// mobject-converters/Converters/REAL_TO_/TryConvert_REAL_TO_UINT
FUNCTION TryConvert_REAL_TO_UINT : BOOL
VAR_INPUT
	in : REAL;
	out : REFERENCE TO UINT;
END_VAR

IF in > DatatypeLimits.MAX_VALUE_OF_REAL_WHICH_CAN_BE_HELD_IN_A_UINT THEN
	RETURN;
END_IF

IF in < DatatypeLimits.MIN_VALUE_OF_REAL_WHICH_CAN_BE_HELD_IN_A_UINT THEN
	RETURN;
END_IF

out := REAL_TO_UINT(in);
TryConvert_REAL_TO_UINT := TRUE;

END_FUNCTION

// mobject-converters/Converters/REAL_TO_/TryConvert_REAL_TO_UDINT
FUNCTION TryConvert_REAL_TO_UDINT : BOOL
VAR_INPUT
	in : REAL;
	out : REFERENCE TO UDINT;
END_VAR

IF in > DatatypeLimits.MAX_VALUE_OF_REAL_WHICH_CAN_BE_HELD_IN_A_UDINT THEN
	RETURN;
END_IF

IF in < DatatypeLimits.MIN_VALUE_OF_REAL_WHICH_CAN_BE_HELD_IN_A_UDINT THEN
	RETURN;
END_IF

out := REAL_TO_UDINT(in);
TryConvert_REAL_TO_UDINT := TRUE;

END_FUNCTION

// mobject-converters/Converters/REAL_TO_/TryConvert_REAL_TO_ULINT
FUNCTION TryConvert_REAL_TO_ULINT : BOOL
VAR_INPUT
	in : REAL;
	out : REFERENCE TO ULINT;
END_VAR

IF in > DatatypeLimits.MAX_VALUE_OF_REAL_WHICH_CAN_BE_HELD_IN_A_ULINT THEN
	RETURN;
END_IF

IF in < DatatypeLimits.MIN_VALUE_OF_REAL_WHICH_CAN_BE_HELD_IN_A_ULINT THEN
	RETURN;
END_IF

out := REAL_TO_ULINT(in);
TryConvert_REAL_TO_ULINT := TRUE;

END_FUNCTION

// mobject-converters/Converters/REAL_TO_/TryConvert_REAL_TO_REAL
FUNCTION TryConvert_REAL_TO_REAL : BOOL
VAR_INPUT
	in : REAL;
	out : REFERENCE TO REAL;
END_VAR

out := in;
TryConvert_REAL_TO_REAL := TRUE;

END_FUNCTION

// mobject-converters/Converters/REAL_TO_/TryConvert_REAL_TO_LREAL
FUNCTION TryConvert_REAL_TO_LREAL : BOOL
VAR_INPUT
	in : REAL;
	out : REFERENCE TO LREAL;
END_VAR

out := REAL_TO_LREAL(in);
TryConvert_REAL_TO_LREAL := TRUE;

END_FUNCTION

// mobject-datatypes/Primitive/_LREAL
{attribute 'linkalways'} 
{attribute 'no_explicit_call' := 'This FB is a CLASS and must be accessed using methods or properties'}
{attribute 'enable_dynamic_creation'}
FUNCTION_BLOCK _LREAL EXTENDS NumericDatatypeBase IMPLEMENTS I_LREAL
VAR
	localData : LREAL;
	activeData : REFERENCE TO LREAL REF= localData;
END_VAR

METHOD FB_init : BOOL
VAR_INPUT
	bInitRetains : BOOL; // if TRUE, the retain variables are initialized (warm start / cold start)
	bInCopyCode : BOOL;  // if TRUE, the instance afterwards gets moved into the copy code (online change)
	InitialValue : LREAL;
END_VAR
localData := InitialValue;
END_METHOD

METHOD PROTECTED SerializeMaxValue
VAR_INPUT
	Serializer : I_Serializer;
END_VAR
Serializer.AddLreal(MaxValue);
END_METHOD

METHOD PROTECTED SerializeMinValue
VAR_INPUT
	Serializer : I_Serializer;
END_VAR
Serializer.AddLreal(MinValue);
END_METHOD

PROPERTY PUBLIC Address : PVOID
GET
Address := ADR(activeData);
END_GET
END_PROPERTY

METHOD PUBLIC ClearReference
VAR_INPUT
END_VAR
activeData REF= localData;
END_METHOD

METHOD PUBLIC Clone : I_Datatype
VAR
    pClone : POINTER TO _LREAL;
END_VAR
pClone := __NEW(_LREAL(InitialValue := Value));
Clone := pClone^;
END_METHOD

PROPERTY PUBLIC IsEven : BOOL
GET
IsEven := FALSE;
END_GET
END_PROPERTY

PROPERTY PUBLIC IsFloat : BOOL
GET
IsFloat := TRUE;
END_GET
END_PROPERTY

PROPERTY PUBLIC IsOdd : BOOL
GET
IsOdd := FALSE;
END_GET
END_PROPERTY

PROPERTY PUBLIC IsSigned : BOOL
GET
IsSigned := TRUE;
END_GET
END_PROPERTY

METHOD PUBLIC MakeReferenceTo
VAR_INPUT
	ReferenceTarget : REFERENCE TO LREAL;
END_VAR
activeData REF= ReferenceTarget;
END_METHOD

PROPERTY PUBLIC MaxValue : LREAL
GET
MaxValue :=  DatatypeLimits.LREAL_MAX_VALUE;
END_GET
END_PROPERTY

PROPERTY PUBLIC MinValue : LREAL
GET
MinValue := DatatypeLimits.LREAL_MIN_VALUE;
END_GET
END_PROPERTY

METHOD PUBLIC SerializeWith
VAR_INPUT
	Serializer : I_Serializer;
END_VAR
Serializer.AddLreal(activeData);
END_METHOD

PROPERTY PUBLIC Size : UDINT
GET
Size := SIZEOF(activeData);
END_GET
END_PROPERTY

METHOD PUBLIC TryConvertTo : BOOL
VAR_INPUT
	Destination : ANY;
END_VAR
TryConvertTo := TryConvert_LREAL_To_Destination(activeData, Destination);
END_METHOD

METHOD PUBLIC TryConvertTo_ : BOOL
VAR_INPUT
	Destination : I_Datatype;
END_VAR
VAR
	resultofBitConversion : BOOL;
	destinationAs_BIT : I_BIT;
	destinationAs_BOOL : I_BOOL;
	destinationAs_BYTE : I_BYTE;
	destinationAs_DINT : I_DINT;
	destinationAs_DT : I_DT;
	destinationAs_DWORD : I_DWORD;
	destinationAs_INT : I_INT;
	destinationAs_LINT : I_LINT;
	destinationAs_LREAL : I_LREAL;
	destinationAs_LWORD : I_LWORD;
	destinationAs_REAL : I_REAL;
	destinationAs_SINT : I_SINT;
	destinationAs_STRING : I_STRING;
	destinationAs_TOD : I_TOD;
	destinationAs_UDINT : I_UDINT;
	destinationAs_UINT : I_UINT;
	destinationAs_ULINT : I_ULINT;
	destinationAs_USINT : I_USINT;
	destinationAs_WORD : I_WORD;
END_VAR
IF destination.TryResolveAs_BIT(destinationAs_BIT) AND_THEN TryConvert_LREAL_TO_BOOL(activeData, resultofBitConversion) THEN
	destinationAs_BIT.Value := resultOfBitConversion;
	TryConvertTo_ := TRUE;
	RETURN;
END_IF

IF destination.TryResolveAs_BOOL(destinationAs_BOOL) THEN
	TryConvertTo_ := TryConvert_LREAL_TO_BOOL(activeData, destinationAs_BOOL.Value);
	RETURN;
END_IF
		
IF destination.TryResolveAs_BYTE(destinationAs_BYTE) THEN
	TryConvertTo_ := TryConvert_LREAL_TO_BYTE(activeData, destinationAs_BYTE.Value);
	RETURN;
END_IF

IF destination.TryResolveAs_DINT(destinationAs_DINT) THEN
	TryConvertTo_ := TryConvert_LREAL_TO_DINT(activeData, destinationAs_DINT.Value);
	RETURN;
END_IF

IF destination.TryResolveAs_DT(destinationAs_DT) THEN
	TryConvertTo_ := TryConvert_LREAL_TO_DT(activeData, destinationAs_DT.Value);
	RETURN;
END_IF

IF destination.TryResolveAs_DWORD(destinationAs_DWORD) THEN
	TryConvertTo_ := TryConvert_LREAL_TO_DWORD(activeData, destinationAs_DWORD.Value);
	RETURN;
END_IF

IF destination.TryResolveAs_INT(destinationAs_INT) THEN
	TryConvertTo_ := TryConvert_LREAL_TO_INT(activeData, destinationAs_INT.Value);
	RETURN;
END_IF

IF destination.TryResolveAs_LINT(destinationAs_LINT) THEN
	TryConvertTo_ := TryConvert_LREAL_TO_LINT(activeData, destinationAs_LINT.Value);
	RETURN;
END_IF

IF destination.TryResolveAs_LREAL(destinationAs_LREAL) THEN
	TryConvertTo_ := TryConvert_LREAL_TO_LREAL(activeData, destinationAs_LREAL.Value);
	RETURN;
END_IF

IF destination.TryResolveAs_LWORD(destinationAs_LWORD) THEN
	TryConvertTo_ := TryConvert_LREAL_TO_LWORD(activeData, destinationAs_LWORD.Value);
	RETURN;
END_IF

IF destination.TryResolveAs_REAL(destinationAs_REAL) THEN
	TryConvertTo_ := TryConvert_LREAL_TO_REAL(activeData, destinationAs_REAL.Value);
	RETURN;
END_IF

IF destination.TryResolveAs_SINT(destinationAs_SINT) THEN
	TryConvertTo_ := TryConvert_LREAL_TO_SINT(activeData, destinationAs_SINT.Value);
	RETURN;
END_IF

IF destination.TryResolveAs_STRING(destinationAs_STRING) THEN
	TryConvertTo_ := TryConvert_LREAL_TO_STRING(activeData, destinationAs_STRING.Value);
	RETURN;
END_IF

IF destination.TryResolveAs_TOD(destinationAs_TOD) THEN
	TryConvertTo_ := TryConvert_LREAL_TO_TOD(activeData, destinationAs_TOD.Value);
	RETURN;
END_IF

IF destination.TryResolveAs_UDINT(destinationAs_UDINT) THEN
	TryConvertTo_ := TryConvert_LREAL_TO_UDINT(activeData, destinationAs_UDINT.Value);
	RETURN;
END_IF

IF destination.TryResolveAs_UINT(destinationAs_UINT) THEN
	TryConvertTo_ := TryConvert_LREAL_TO_UINT(activeData, destinationAs_UINT.Value);
	RETURN;
END_IF

IF destination.TryResolveAs_ULINT(destinationAs_ULINT) THEN
	TryConvertTo_ := TryConvert_LREAL_TO_ULINT(activeData, destinationAs_ULINT.Value);
	RETURN;
END_IF

IF destination.TryResolveAs_USINT(destinationAs_USINT) THEN
	TryConvertTo_ := TryConvert_LREAL_TO_USINT(activeData, destinationAs_USINT.Value);
	RETURN;
END_IF

IF destination.TryResolveAs_WORD(destinationAs_WORD) THEN
	TryConvertTo_ := TryConvert_LREAL_TO_WORD(activeData, destinationAs_WORD.Value);
	RETURN;
END_IF
END_METHOD

METHOD TryDeserializeFrom : BOOL
VAR_INPUT
	Deserializer : I_Deserializer;
	Feedback : I_DeserializerFeedback;
END_VAR
TryDeserializeFrom := Deserializer.TryGetLreal(activeData, Feedback);
END_METHOD

METHOD TryMakeReferenceTo : BOOL
VAR_INPUT
	Target : I_Datatype;
END_VAR
VAR
	pTargetData : POINTER TO LREAL;
END_VAR
IF NOT IsEquivalentTo(Target) THEN
	RETURN;
END_IF

pTargetData := Target.Address;
activeData REF= pTargetData^;
TryMakeReferenceTo := TRUE;
END_METHOD

METHOD PUBLIC TryResolveAs_LREAL : BOOL
VAR_INPUT
	Destination : REFERENCE TO I_LREAL;
END_VAR
Destination := THIS^;
TryResolveAs_LREAL := TRUE;
END_METHOD

PROPERTY PUBLIC TypeName : T_MAXSTRING
GET
TypeName := 'LREAL';
END_GET
END_PROPERTY

{warning disable C5410}
PROPERTY PUBLIC Value : REFERENCE TO LREAL
{warning restore C5410}
GET
Value REF= activeData;
END_GET
END_PROPERTY

END_FUNCTION_BLOCK

// mobject-converters/Converters/LREAL_TO_/TryConvert_LREAL_TO_Destination
FUNCTION TryConvert_LREAL_TO_Destination : BOOL
VAR_INPUT
	in : LREAL;
	out : ANY;
END_VAR
VAR
	convertResult : BOOL := FALSE;
	convertAddress : PVOID;
	_BOOL : BOOL;
	_BYTE : BYTE;
	_WORD : WORD;
	_DWORD : DWORD;
	_LWORD : LWORD;
	_SINT : SINT;
	_INT : INT;
	_DINT : DINT;
	_LINT : LINT;
	_USINT : USINT;
	_UINT : UINT;
	_UDINT : UDINT;
	_ULINT : ULINT;
	_REAL : REAL;
	_LREAL : LREAL;
	_TIME : TIME;
	_TOD : TOD;
	_DATE : DATE;
	_DT : DT;
	_STRING : STRING;
END_VAR

CASE out.TypeClass OF
	__SYSTEM.TYPE_CLASS.TYPE_BOOL:
	
	convertResult := TryConvert_LREAL_TO_BOOL(in, _BOOL);
	IF convertResult THEN
		convertAddress := ADR(_BOOL);
	END_IF
	
	__SYSTEM.TYPE_CLASS.TYPE_BYTE:
	
	convertResult := TryConvert_LREAL_TO_BYTE(in, _BYTE);
	IF convertResult THEN
		convertAddress := ADR(_BYTE);
	END_IF
	
	__SYSTEM.TYPE_CLASS.TYPE_WORD:
	
	convertResult := TryConvert_LREAL_TO_WORD(in, _WORD);
	IF convertResult THEN
		convertAddress := ADR(_WORD);
	END_IF
	
	__SYSTEM.TYPE_CLASS.TYPE_DWORD:
	
	convertResult := TryConvert_LREAL_TO_DWORD(in, _DWORD);
	IF convertResult THEN
		convertAddress := ADR(_DWORD);
	END_IF
	
	__SYSTEM.TYPE_CLASS.TYPE_LWORD:
	
	convertResult := TryConvert_LREAL_TO_LWORD(in, _LWORD);
	IF convertResult THEN
		convertAddress := ADR(_LWORD);
	END_IF
	
	__SYSTEM.TYPE_CLASS.TYPE_SINT:
	
	convertResult := TryConvert_LREAL_TO_SINT(in, _SINT);
	IF convertResult THEN
		convertAddress := ADR(_SINT);
	END_IF
	
	__SYSTEM.TYPE_CLASS.TYPE_INT:
	
	convertResult := TryConvert_LREAL_TO_INT(in, _INT);
	IF convertResult THEN
		convertAddress := ADR(_INT);
	END_IF
	
	__SYSTEM.TYPE_CLASS.TYPE_DINT:
	
	convertResult := TryConvert_LREAL_TO_DINT(in, _DINT);
	IF convertResult THEN
		convertAddress := ADR(_DINT);
	END_IF
	
	__SYSTEM.TYPE_CLASS.TYPE_LINT:
	
	convertResult := TryConvert_LREAL_TO_LINT(in, _LINT);
	IF convertResult THEN
		convertAddress := ADR(_LINT);
	END_IF
	
	__SYSTEM.TYPE_CLASS.TYPE_USINT:
	
	convertResult := TryConvert_LREAL_TO_USINT(in, _USINT);
	IF convertResult THEN
		convertAddress := ADR(_USINT);
	END_IF
	
	__SYSTEM.TYPE_CLASS.TYPE_UINT:
	
	convertResult := TryConvert_LREAL_TO_UINT(in, _UINT);
	IF convertResult THEN
		convertAddress := ADR(_UINT);
	END_IF
	
	__SYSTEM.TYPE_CLASS.TYPE_UDINT:
	
	convertResult := TryConvert_LREAL_TO_UDINT(in, _UDINT);
	IF convertResult THEN
		convertAddress := ADR(_UDINT);
	END_IF
	
	__SYSTEM.TYPE_CLASS.TYPE_ULINT:
	
	convertResult := TryConvert_LREAL_TO_ULINT(in, _ULINT);
	IF convertResult THEN
		convertAddress := ADR(_ULINT);
	END_IF
	
	__SYSTEM.TYPE_CLASS.TYPE_REAL:
	
	convertResult := TryConvert_LREAL_TO_REAL(in, _REAL);
	IF convertResult THEN
		convertAddress := ADR(_REAL);
	END_IF
	
	__SYSTEM.TYPE_CLASS.TYPE_LREAL:
	
	convertResult := TryConvert_LREAL_TO_LREAL(in, _LREAL);
	IF convertResult THEN
		convertAddress := ADR(_LREAL);
	END_IF
	
	__SYSTEM.TYPE_CLASS.TYPE_TIME:
	
	convertResult := TryConvert_LREAL_TO_TIME(in, _TIME);
	IF convertResult THEN
		convertAddress := ADR(_TIME);
	END_IF
	
	__SYSTEM.TYPE_CLASS.TYPE_TIMEOFDAY:
	
	convertResult := TryConvert_LREAL_TO_TOD(in, _TOD);
	IF convertResult THEN
		convertAddress := ADR(_TOD);
	END_IF
	
	__SYSTEM.TYPE_CLASS.TYPE_DATE:
	
	convertResult := TryConvert_LREAL_TO_DATE(in, _DATE);
	IF convertResult THEN
		convertAddress := ADR(_DATE);
	END_IF
	
	__SYSTEM.TYPE_CLASS.TYPE_DATEANDTIME:
	
	convertResult := TryConvert_LREAL_TO_DT(in, _DT);
	IF convertResult THEN
		convertAddress := ADR(_DT);
	END_IF
	
	__SYSTEM.TYPE_CLASS.TYPE_STRING:
	
	convertResult := TryConvert_LREAL_TO_STRING(in, _STRING);
	IF convertResult THEN
		convertAddress := ADR(_STRING);
	END_IF
	
END_CASE

IF convertResult THEN
	memcpy(out.pValue,convertAddress,DINT_TO_UDINT(out.diSize));
END_IF

TryConvert_LREAL_TO_Destination := convertResult;

END_FUNCTION

// mobject-converters/Converters/LREAL_TO_/TryConvert_LREAL_TO_BOOL
FUNCTION TryConvert_LREAL_TO_BOOL : BOOL
VAR_INPUT
	in : LREAL;
	out : REFERENCE TO BOOL;
END_VAR

out := LREAL_TO_BOOL(in);
TryConvert_LREAL_TO_BOOL := TRUE;

END_FUNCTION

// mobject-converters/Converters/LREAL_TO_/TryConvert_LREAL_TO_BYTE
FUNCTION TryConvert_LREAL_TO_BYTE : BOOL
VAR_INPUT
	in : LREAL;
	out : REFERENCE TO BYTE;
END_VAR

IF in > DatatypeLimits.MAX_VALUE_OF_LREAL_WHICH_CAN_BE_HELD_IN_A_BYTE THEN
	RETURN;
END_IF

IF in < DatatypeLimits.MIN_VALUE_OF_LREAL_WHICH_CAN_BE_HELD_IN_A_BYTE THEN
	RETURN;
END_IF

out := LREAL_TO_BYTE(in);
TryConvert_LREAL_TO_BYTE := TRUE;

END_FUNCTION

// mobject-converters/Converters/LREAL_TO_/TryConvert_LREAL_TO_WORD
FUNCTION TryConvert_LREAL_TO_WORD : BOOL
VAR_INPUT
	in : LREAL;
	out : REFERENCE TO WORD;
END_VAR

IF in > DatatypeLimits.MAX_VALUE_OF_LREAL_WHICH_CAN_BE_HELD_IN_A_WORD THEN
	RETURN;
END_IF

IF in < DatatypeLimits.MIN_VALUE_OF_LREAL_WHICH_CAN_BE_HELD_IN_A_WORD THEN
	RETURN;
END_IF

out := LREAL_TO_WORD(in);
TryConvert_LREAL_TO_WORD := TRUE;

END_FUNCTION

// mobject-converters/Converters/LREAL_TO_/TryConvert_LREAL_TO_DWORD
FUNCTION TryConvert_LREAL_TO_DWORD : BOOL
VAR_INPUT
	in : LREAL;
	out : REFERENCE TO DWORD;
END_VAR

IF in > DatatypeLimits.MAX_VALUE_OF_LREAL_WHICH_CAN_BE_HELD_IN_A_DWORD THEN
	RETURN;
END_IF

IF in < DatatypeLimits.MIN_VALUE_OF_LREAL_WHICH_CAN_BE_HELD_IN_A_DWORD THEN
	RETURN;
END_IF

out := LREAL_TO_DWORD(in);
TryConvert_LREAL_TO_DWORD := TRUE;

END_FUNCTION

// mobject-converters/Converters/LREAL_TO_/TryConvert_LREAL_TO_LWORD
FUNCTION TryConvert_LREAL_TO_LWORD : BOOL
VAR_INPUT
	in : LREAL;
	out : REFERENCE TO LWORD;
END_VAR

IF in > DatatypeLimits.MAX_VALUE_OF_LREAL_WHICH_CAN_BE_HELD_IN_A_LWORD THEN
	RETURN;
END_IF

IF in < DatatypeLimits.MIN_VALUE_OF_LREAL_WHICH_CAN_BE_HELD_IN_A_LWORD THEN
	RETURN;
END_IF

out := LREAL_TO_LWORD(in);
TryConvert_LREAL_TO_LWORD := TRUE;

END_FUNCTION

// mobject-converters/Converters/LREAL_TO_/TryConvert_LREAL_TO_SINT
FUNCTION TryConvert_LREAL_TO_SINT : BOOL
VAR_INPUT
	in : LREAL;
	out : REFERENCE TO SINT;
END_VAR

IF in > DatatypeLimits.MAX_VALUE_OF_LREAL_WHICH_CAN_BE_HELD_IN_A_SINT THEN
	RETURN;
END_IF

IF in < DatatypeLimits.MIN_VALUE_OF_LREAL_WHICH_CAN_BE_HELD_IN_A_SINT THEN
	RETURN;
END_IF

out := LREAL_TO_SINT(in);
TryConvert_LREAL_TO_SINT := TRUE;

END_FUNCTION

// mobject-converters/Converters/LREAL_TO_/TryConvert_LREAL_TO_INT
FUNCTION TryConvert_LREAL_TO_INT : BOOL
VAR_INPUT
	in : LREAL;
	out : REFERENCE TO INT;
END_VAR

IF in > DatatypeLimits.MAX_VALUE_OF_LREAL_WHICH_CAN_BE_HELD_IN_A_INT THEN
	RETURN;
END_IF

IF in < DatatypeLimits.MIN_VALUE_OF_LREAL_WHICH_CAN_BE_HELD_IN_A_INT THEN
	RETURN;
END_IF

out := LREAL_TO_INT(in);
TryConvert_LREAL_TO_INT := TRUE;

END_FUNCTION

// mobject-converters/Converters/LREAL_TO_/TryConvert_LREAL_TO_DINT
FUNCTION TryConvert_LREAL_TO_DINT : BOOL
VAR_INPUT
	in : LREAL;
	out : REFERENCE TO DINT;
END_VAR

IF in > DatatypeLimits.MAX_VALUE_OF_LREAL_WHICH_CAN_BE_HELD_IN_A_DINT THEN
	RETURN;
END_IF

IF in < DatatypeLimits.MIN_VALUE_OF_LREAL_WHICH_CAN_BE_HELD_IN_A_DINT THEN
	RETURN;
END_IF

out := LREAL_TO_DINT(in);
TryConvert_LREAL_TO_DINT := TRUE;

END_FUNCTION

// mobject-converters/Converters/LREAL_TO_/TryConvert_LREAL_TO_LINT
FUNCTION TryConvert_LREAL_TO_LINT : BOOL
VAR_INPUT
	in : LREAL;
	out : REFERENCE TO LINT;
END_VAR

IF in > DatatypeLimits.MAX_VALUE_OF_LREAL_WHICH_CAN_BE_HELD_IN_A_LINT THEN
	RETURN;
END_IF

IF in < DatatypeLimits.MIN_VALUE_OF_LREAL_WHICH_CAN_BE_HELD_IN_A_LINT THEN
	RETURN;
END_IF

out := LREAL_TO_LINT(in);
TryConvert_LREAL_TO_LINT := TRUE;

END_FUNCTION

// mobject-converters/Converters/LREAL_TO_/TryConvert_LREAL_TO_USINT
FUNCTION TryConvert_LREAL_TO_USINT : BOOL
VAR_INPUT
	in : LREAL;
	out : REFERENCE TO USINT;
END_VAR

IF in > DatatypeLimits.MAX_VALUE_OF_LREAL_WHICH_CAN_BE_HELD_IN_A_USINT THEN
	RETURN;
END_IF

IF in < DatatypeLimits.MIN_VALUE_OF_LREAL_WHICH_CAN_BE_HELD_IN_A_USINT THEN
	RETURN;
END_IF

out := LREAL_TO_USINT(in);
TryConvert_LREAL_TO_USINT := TRUE;

END_FUNCTION

// mobject-converters/Converters/LREAL_TO_/TryConvert_LREAL_TO_UINT
FUNCTION TryConvert_LREAL_TO_UINT : BOOL
VAR_INPUT
	in : LREAL;
	out : REFERENCE TO UINT;
END_VAR

IF in > DatatypeLimits.MAX_VALUE_OF_LREAL_WHICH_CAN_BE_HELD_IN_A_UINT THEN
	RETURN;
END_IF

IF in < DatatypeLimits.MIN_VALUE_OF_LREAL_WHICH_CAN_BE_HELD_IN_A_UINT THEN
	RETURN;
END_IF

out := LREAL_TO_UINT(in);
TryConvert_LREAL_TO_UINT := TRUE;

END_FUNCTION

// mobject-converters/Converters/LREAL_TO_/TryConvert_LREAL_TO_UDINT
FUNCTION TryConvert_LREAL_TO_UDINT : BOOL
VAR_INPUT
	in : LREAL;
	out : REFERENCE TO UDINT;
END_VAR

IF in > DatatypeLimits.MAX_VALUE_OF_LREAL_WHICH_CAN_BE_HELD_IN_A_UDINT THEN
	RETURN;
END_IF

IF in < DatatypeLimits.MIN_VALUE_OF_LREAL_WHICH_CAN_BE_HELD_IN_A_UDINT THEN
	RETURN;
END_IF

out := LREAL_TO_UDINT(in);
TryConvert_LREAL_TO_UDINT := TRUE;

END_FUNCTION

// mobject-converters/Converters/LREAL_TO_/TryConvert_LREAL_TO_ULINT
FUNCTION TryConvert_LREAL_TO_ULINT : BOOL
VAR_INPUT
	in : LREAL;
	out : REFERENCE TO ULINT;
END_VAR

IF in > DatatypeLimits.MAX_VALUE_OF_LREAL_WHICH_CAN_BE_HELD_IN_A_ULINT THEN
	RETURN;
END_IF

IF in < DatatypeLimits.MIN_VALUE_OF_LREAL_WHICH_CAN_BE_HELD_IN_A_ULINT THEN
	RETURN;
END_IF

out := LREAL_TO_ULINT(in);
TryConvert_LREAL_TO_ULINT := TRUE;

END_FUNCTION

// mobject-converters/Converters/LREAL_TO_/TryConvert_LREAL_TO_REAL
FUNCTION TryConvert_LREAL_TO_REAL : BOOL
VAR_INPUT
	in : LREAL;
	out : REFERENCE TO REAL;
END_VAR

IF in > DatatypeLimits.MAX_VALUE_OF_LREAL_WHICH_CAN_BE_HELD_IN_A_REAL THEN
	RETURN;
END_IF

IF in < DatatypeLimits.MIN_VALUE_OF_LREAL_WHICH_CAN_BE_HELD_IN_A_REAL THEN
	RETURN;
END_IF

out := LREAL_TO_REAL(in);
TryConvert_LREAL_TO_REAL := TRUE;

END_FUNCTION

// mobject-converters/Converters/LREAL_TO_/TryConvert_LREAL_TO_LREAL
FUNCTION TryConvert_LREAL_TO_LREAL : BOOL
VAR_INPUT
	in : LREAL;
	out : REFERENCE TO LREAL;
END_VAR

out := in;
TryConvert_LREAL_TO_LREAL := TRUE;

END_FUNCTION

// mobject-converters/Converters/LREAL_TO_/TryConvert_LREAL_TO_TIME
FUNCTION TryConvert_LREAL_TO_TIME : BOOL
VAR_INPUT
	in : LREAL;
	out : REFERENCE TO TIME;
END_VAR

IF in > DatatypeLimits.MAX_VALUE_OF_LREAL_WHICH_CAN_BE_HELD_IN_A_TIME THEN
	RETURN;
END_IF

IF in < DatatypeLimits.MIN_VALUE_OF_LREAL_WHICH_CAN_BE_HELD_IN_A_TIME THEN
	RETURN;
END_IF

out := LREAL_TO_TIME(in);
TryConvert_LREAL_TO_TIME := TRUE;

END_FUNCTION

// mobject-converters/Converters/LREAL_TO_/TryConvert_LREAL_TO_TOD
FUNCTION TryConvert_LREAL_TO_TOD : BOOL
VAR_INPUT
	in : LREAL;
	out : REFERENCE TO TOD;
END_VAR

IF in > DatatypeLimits.MAX_VALUE_OF_LREAL_WHICH_CAN_BE_HELD_IN_A_TOD THEN
	RETURN;
END_IF

IF in < DatatypeLimits.MIN_VALUE_OF_LREAL_WHICH_CAN_BE_HELD_IN_A_TOD THEN
	RETURN;
END_IF

out := LREAL_TO_TOD(in);
TryConvert_LREAL_TO_TOD := TRUE;

END_FUNCTION

// mobject-datatypes/Primitive/_TOD
{attribute 'linkalways'} 
{attribute 'no_explicit_call' := 'This FB is a CLASS and must be accessed using methods or properties'}
{attribute 'enable_dynamic_creation'}
FUNCTION_BLOCK _TOD EXTENDS DatatypeBase IMPLEMENTS I_TOD
VAR
	localData : TOD;
	activeData : REFERENCE TO TOD REF= localData;
END_VAR

METHOD FB_init : BOOL
VAR_INPUT
	bInitRetains : BOOL; // if TRUE, the retain variables are initialized (warm start / cold start)
	bInCopyCode : BOOL;  // if TRUE, the instance afterwards gets moved WORDo the copy code (online change)
	InitialValue : TOD;
END_VAR
localData := InitialValue;
END_METHOD

PROPERTY PUBLIC Address : PVOID
GET
Address := ADR(activeData);
END_GET
END_PROPERTY

METHOD PUBLIC ClearReference
VAR_INPUT
END_VAR
activeData REF= localData;
END_METHOD

METHOD PUBLIC Clone : I_Datatype
VAR
    pClone : POINTER TO _TOD;
END_VAR
pClone := __NEW(_TOD(InitialValue := Value));
Clone := pClone^;
END_METHOD

METHOD PUBLIC MakeReferenceTo
VAR_INPUT
	ReferenceTarget : REFERENCE TO TOD;
END_VAR
activeData REF= ReferenceTarget;
END_METHOD

METHOD PUBLIC SerializeWith
VAR_INPUT
	Serializer : I_Serializer;
END_VAR
Serializer.AddTod(activeData);
END_METHOD

PROPERTY PUBLIC Size : UDINT
GET
Size := SIZEOF(activeData);
END_GET
END_PROPERTY

METHOD PUBLIC TryConvertTo : BOOL
VAR_INPUT
	Destination : ANY;
END_VAR
TryConvertTo := TryConvert_TOD_TO_Destination(activeData, Destination);
END_METHOD

METHOD PUBLIC TryConvertTo_ : BOOL
VAR_INPUT
	Destination : I_Datatype;
END_VAR
VAR
	resultofBitConversion : BOOL;
	destinationAs_BIT : I_BIT;
	destinationAs_BOOL : I_BOOL;
	destinationAs_BYTE : I_BYTE;
	destinationAs_DINT : I_DINT;
	destinationAs_DT : I_DT;
	destinationAs_DWORD : I_DWORD;
	destinationAs_INT : I_INT;
	destinationAs_LINT : I_LINT;
	destinationAs_LREAL : I_LREAL;
	destinationAs_LWORD : I_LWORD;
	destinationAs_REAL : I_REAL;
	destinationAs_SINT : I_SINT;
	destinationAs_STRING : I_STRING;
	destinationAs_TOD : I_TOD;
	destinationAs_UDINT : I_UDINT;
	destinationAs_UINT : I_UINT;
	destinationAs_ULINT : I_ULINT;
	destinationAs_USINT : I_USINT;
	destinationAs_WORD : I_WORD;
END_VAR
IF destination.TryResolveAs_BIT(destinationAs_BIT) AND_THEN TryConvert_TOD_TO_BOOL(activeData, resultofBitConversion) THEN
	destinationAs_BIT.Value := resultOfBitConversion;
	TryConvertTo_ := TRUE;
	RETURN;
END_IF

IF destination.TryResolveAs_BOOL(destinationAs_BOOL) THEN
	TryConvertTo_ := TryConvert_TOD_TO_BOOL(activeData, destinationAs_BOOL.Value);
	RETURN;
END_IF
		
IF destination.TryResolveAs_BYTE(destinationAs_BYTE) THEN
	TryConvertTo_ := TryConvert_TOD_TO_BYTE(activeData, destinationAs_BYTE.Value);
	RETURN;
END_IF

IF destination.TryResolveAs_DINT(destinationAs_DINT) THEN
	TryConvertTo_ := TryConvert_TOD_TO_DINT(activeData, destinationAs_DINT.Value);
	RETURN;
END_IF

IF destination.TryResolveAs_DT(destinationAs_DT) THEN
	TryConvertTo_ := TryConvert_TOD_TO_DT(activeData, destinationAs_DT.Value);
	RETURN;
END_IF

IF destination.TryResolveAs_DWORD(destinationAs_DWORD) THEN
	TryConvertTo_ := TryConvert_TOD_TO_DWORD(activeData, destinationAs_DWORD.Value);
	RETURN;
END_IF

IF destination.TryResolveAs_INT(destinationAs_INT) THEN
	TryConvertTo_ := TryConvert_TOD_TO_INT(activeData, destinationAs_INT.Value);
	RETURN;
END_IF

IF destination.TryResolveAs_LINT(destinationAs_LINT) THEN
	TryConvertTo_ := TryConvert_TOD_TO_LINT(activeData, destinationAs_LINT.Value);
	RETURN;
END_IF

IF destination.TryResolveAs_LREAL(destinationAs_LREAL) THEN
	TryConvertTo_ := TryConvert_TOD_TO_LREAL(activeData, destinationAs_LREAL.Value);
	RETURN;
END_IF

IF destination.TryResolveAs_LWORD(destinationAs_LWORD) THEN
	TryConvertTo_ := TryConvert_TOD_TO_LWORD(activeData, destinationAs_LWORD.Value);
	RETURN;
END_IF

IF destination.TryResolveAs_REAL(destinationAs_REAL) THEN
	TryConvertTo_ := TryConvert_TOD_TO_REAL(activeData, destinationAs_REAL.Value);
	RETURN;
END_IF

IF destination.TryResolveAs_SINT(destinationAs_SINT) THEN
	TryConvertTo_ := TryConvert_TOD_TO_SINT(activeData, destinationAs_SINT.Value);
	RETURN;
END_IF

IF destination.TryResolveAs_STRING(destinationAs_STRING) THEN
	TryConvertTo_ := TryConvert_TOD_TO_STRING(activeData, destinationAs_STRING.Value);
	RETURN;
END_IF

IF destination.TryResolveAs_TOD(destinationAs_TOD) THEN
	TryConvertTo_ := TryConvert_TOD_TO_TOD(activeData, destinationAs_TOD.Value);
	RETURN;
END_IF

IF destination.TryResolveAs_UDINT(destinationAs_UDINT) THEN
	TryConvertTo_ := TryConvert_TOD_TO_UDINT(activeData, destinationAs_UDINT.Value);
	RETURN;
END_IF

IF destination.TryResolveAs_UINT(destinationAs_UINT) THEN
	TryConvertTo_ := TryConvert_TOD_TO_UINT(activeData, destinationAs_UINT.Value);
	RETURN;
END_IF

IF destination.TryResolveAs_ULINT(destinationAs_ULINT) THEN
	TryConvertTo_ := TryConvert_TOD_TO_ULINT(activeData, destinationAs_ULINT.Value);
	RETURN;
END_IF

IF destination.TryResolveAs_USINT(destinationAs_USINT) THEN
	TryConvertTo_ := TryConvert_TOD_TO_USINT(activeData, destinationAs_USINT.Value);
	RETURN;
END_IF

IF destination.TryResolveAs_WORD(destinationAs_WORD) THEN
	TryConvertTo_ := TryConvert_TOD_TO_WORD(activeData, destinationAs_WORD.Value);
	RETURN;
END_IF
END_METHOD

METHOD TryDeserializeFrom : BOOL
VAR_INPUT
	Deserializer : I_Deserializer;
	Feedback : I_DeserializerFeedback;
END_VAR
TryDeserializeFrom := Deserializer.TryGetTod(activeData, Feedback);
END_METHOD

METHOD TryMakeReferenceTo : BOOL
VAR_INPUT
	Target : I_Datatype;
END_VAR
VAR
	pTargetData : POINTER TO TOD;
END_VAR
IF NOT IsEquivalentTo(Target) THEN
	RETURN;
END_IF

pTargetData := Target.Address;
activeData REF= pTargetData^;
TryMakeReferenceTo := TRUE;
END_METHOD

METHOD PUBLIC TryResolveAs_TOD : BOOL
VAR_INPUT
	Destination : REFERENCE TO I_TOD;
END_VAR
Destination := THIS^;
TryResolveAs_TOD := TRUE;
END_METHOD

PROPERTY PUBLIC TypeName : T_MAXSTRING
GET
TypeName := 'TOD';
END_GET
END_PROPERTY

{warning disable C5410}
PROPERTY PUBLIC Value : REFERENCE TO TOD
{warning restore C5410}
GET
Value REF= activeData;
END_GET
END_PROPERTY

END_FUNCTION_BLOCK

// mobject-converters/Converters/TOD_TO_/TryConvert_TOD_TO_Destination
FUNCTION TryConvert_TOD_TO_Destination : BOOL
VAR_INPUT
	in : TOD;
	out : ANY;
END_VAR
VAR
	convertResult : BOOL := FALSE;
	convertAddress : PVOID;
	_BOOL : BOOL;
	_BYTE : BYTE;
	_WORD : WORD;
	_DWORD : DWORD;
	_LWORD : LWORD;
	_SINT : SINT;
	_INT : INT;
	_DINT : DINT;
	_LINT : LINT;
	_USINT : USINT;
	_UINT : UINT;
	_UDINT : UDINT;
	_ULINT : ULINT;
	_REAL : REAL;
	_LREAL : LREAL;
	_TIME : TIME;
	_TOD : TOD;
	_DATE : DATE;
	_DT : DT;
	_STRING : STRING;
END_VAR

CASE out.TypeClass OF
	__SYSTEM.TYPE_CLASS.TYPE_BOOL:
	
	convertResult := TryConvert_TOD_TO_BOOL(in, _BOOL);
	IF convertResult THEN
		convertAddress := ADR(_BOOL);
	END_IF
	
	__SYSTEM.TYPE_CLASS.TYPE_BYTE:
	
	convertResult := TryConvert_TOD_TO_BYTE(in, _BYTE);
	IF convertResult THEN
		convertAddress := ADR(_BYTE);
	END_IF
	
	__SYSTEM.TYPE_CLASS.TYPE_WORD:
	
	convertResult := TryConvert_TOD_TO_WORD(in, _WORD);
	IF convertResult THEN
		convertAddress := ADR(_WORD);
	END_IF
	
	__SYSTEM.TYPE_CLASS.TYPE_DWORD:
	
	convertResult := TryConvert_TOD_TO_DWORD(in, _DWORD);
	IF convertResult THEN
		convertAddress := ADR(_DWORD);
	END_IF
	
	__SYSTEM.TYPE_CLASS.TYPE_LWORD:
	
	convertResult := TryConvert_TOD_TO_LWORD(in, _LWORD);
	IF convertResult THEN
		convertAddress := ADR(_LWORD);
	END_IF
	
	__SYSTEM.TYPE_CLASS.TYPE_SINT:
	
	convertResult := TryConvert_TOD_TO_SINT(in, _SINT);
	IF convertResult THEN
		convertAddress := ADR(_SINT);
	END_IF
	
	__SYSTEM.TYPE_CLASS.TYPE_INT:
	
	convertResult := TryConvert_TOD_TO_INT(in, _INT);
	IF convertResult THEN
		convertAddress := ADR(_INT);
	END_IF
	
	__SYSTEM.TYPE_CLASS.TYPE_DINT:
	
	convertResult := TryConvert_TOD_TO_DINT(in, _DINT);
	IF convertResult THEN
		convertAddress := ADR(_DINT);
	END_IF
	
	__SYSTEM.TYPE_CLASS.TYPE_LINT:
	
	convertResult := TryConvert_TOD_TO_LINT(in, _LINT);
	IF convertResult THEN
		convertAddress := ADR(_LINT);
	END_IF
	
	__SYSTEM.TYPE_CLASS.TYPE_USINT:
	
	convertResult := TryConvert_TOD_TO_USINT(in, _USINT);
	IF convertResult THEN
		convertAddress := ADR(_USINT);
	END_IF
	
	__SYSTEM.TYPE_CLASS.TYPE_UINT:
	
	convertResult := TryConvert_TOD_TO_UINT(in, _UINT);
	IF convertResult THEN
		convertAddress := ADR(_UINT);
	END_IF
	
	__SYSTEM.TYPE_CLASS.TYPE_UDINT:
	
	convertResult := TryConvert_TOD_TO_UDINT(in, _UDINT);
	IF convertResult THEN
		convertAddress := ADR(_UDINT);
	END_IF
	
	__SYSTEM.TYPE_CLASS.TYPE_ULINT:
	
	convertResult := TryConvert_TOD_TO_ULINT(in, _ULINT);
	IF convertResult THEN
		convertAddress := ADR(_ULINT);
	END_IF
	
	__SYSTEM.TYPE_CLASS.TYPE_REAL:
	
	convertResult := TryConvert_TOD_TO_REAL(in, _REAL);
	IF convertResult THEN
		convertAddress := ADR(_REAL);
	END_IF
	
	__SYSTEM.TYPE_CLASS.TYPE_LREAL:
	
	convertResult := TryConvert_TOD_TO_LREAL(in, _LREAL);
	IF convertResult THEN
		convertAddress := ADR(_LREAL);
	END_IF
	
	__SYSTEM.TYPE_CLASS.TYPE_TIME:
	
	convertResult := TryConvert_TOD_TO_TIME(in, _TIME);
	IF convertResult THEN
		convertAddress := ADR(_TIME);
	END_IF
	
	__SYSTEM.TYPE_CLASS.TYPE_TIMEOFDAY:
	
	convertResult := TryConvert_TOD_TO_TOD(in, _TOD);
	IF convertResult THEN
		convertAddress := ADR(_TOD);
	END_IF
	
	__SYSTEM.TYPE_CLASS.TYPE_DATE:
	
	convertResult := TryConvert_TOD_TO_DATE(in, _DATE);
	IF convertResult THEN
		convertAddress := ADR(_DATE);
	END_IF
	
	__SYSTEM.TYPE_CLASS.TYPE_DATEANDTIME:
	
	convertResult := TryConvert_TOD_TO_DT(in, _DT);
	IF convertResult THEN
		convertAddress := ADR(_DT);
	END_IF
	
	__SYSTEM.TYPE_CLASS.TYPE_STRING:
	
	convertResult := TryConvert_TOD_TO_STRING(in, _STRING);
	IF convertResult THEN
		convertAddress := ADR(_STRING);
	END_IF
	
END_CASE

IF convertResult THEN
	memcpy(out.pValue,convertAddress,DINT_TO_UDINT(out.diSize));
END_IF

TryConvert_TOD_TO_Destination := convertResult;

END_FUNCTION

// mobject-converters/Converters/TOD_TO_/TryConvert_TOD_TO_BOOL
FUNCTION TryConvert_TOD_TO_BOOL : BOOL
VAR_INPUT
	in : TOD;
	out : REFERENCE TO BOOL;
END_VAR

out := TOD_TO_BOOL(in);
TryConvert_TOD_TO_BOOL := TRUE;

END_FUNCTION

// mobject-converters/Converters/TOD_TO_/TryConvert_TOD_TO_BYTE
FUNCTION TryConvert_TOD_TO_BYTE : BOOL
VAR_INPUT
	in : TOD;
	out : REFERENCE TO BYTE;
END_VAR

IF in > DatatypeLimits.MAX_VALUE_OF_TOD_WHICH_CAN_BE_HELD_IN_A_BYTE THEN
	RETURN;
END_IF

out := TOD_TO_BYTE(in);
TryConvert_TOD_TO_BYTE := TRUE;

END_FUNCTION

// mobject-converters/Converters/TOD_TO_/TryConvert_TOD_TO_WORD
FUNCTION TryConvert_TOD_TO_WORD : BOOL
VAR_INPUT
	in : TOD;
	out : REFERENCE TO WORD;
END_VAR

IF in > DatatypeLimits.MAX_VALUE_OF_TOD_WHICH_CAN_BE_HELD_IN_A_WORD THEN
	RETURN;
END_IF

out := TOD_TO_WORD(in);
TryConvert_TOD_TO_WORD := TRUE;

END_FUNCTION

// mobject-converters/Converters/TOD_TO_/TryConvert_TOD_TO_DWORD
FUNCTION TryConvert_TOD_TO_DWORD : BOOL
VAR_INPUT
	in : TOD;
	out : REFERENCE TO DWORD;
END_VAR

out := TOD_TO_DWORD(in);
TryConvert_TOD_TO_DWORD := TRUE;

END_FUNCTION

// mobject-converters/Converters/TOD_TO_/TryConvert_TOD_TO_LWORD
FUNCTION TryConvert_TOD_TO_LWORD : BOOL
VAR_INPUT
	in : TOD;
	out : REFERENCE TO LWORD;
END_VAR

out := TOD_TO_LWORD(in);
TryConvert_TOD_TO_LWORD := TRUE;

END_FUNCTION

// mobject-converters/Converters/TOD_TO_/TryConvert_TOD_TO_SINT
FUNCTION TryConvert_TOD_TO_SINT : BOOL
VAR_INPUT
	in : TOD;
	out : REFERENCE TO SINT;
END_VAR

IF in > DatatypeLimits.MAX_VALUE_OF_TOD_WHICH_CAN_BE_HELD_IN_A_SINT THEN
	RETURN;
END_IF

out := TOD_TO_SINT(in);
TryConvert_TOD_TO_SINT := TRUE;

END_FUNCTION

// mobject-converters/Converters/TOD_TO_/TryConvert_TOD_TO_INT
FUNCTION TryConvert_TOD_TO_INT : BOOL
VAR_INPUT
	in : TOD;
	out : REFERENCE TO INT;
END_VAR

IF in > DatatypeLimits.MAX_VALUE_OF_TOD_WHICH_CAN_BE_HELD_IN_A_INT THEN
	RETURN;
END_IF

out := TOD_TO_INT(in);
TryConvert_TOD_TO_INT := TRUE;

END_FUNCTION

// mobject-converters/Converters/TOD_TO_/TryConvert_TOD_TO_DINT
FUNCTION TryConvert_TOD_TO_DINT : BOOL
VAR_INPUT
	in : TOD;
	out : REFERENCE TO DINT;
END_VAR

out := TOD_TO_DINT(in);
TryConvert_TOD_TO_DINT := TRUE;

END_FUNCTION

// mobject-converters/Converters/TOD_TO_/TryConvert_TOD_TO_LINT
FUNCTION TryConvert_TOD_TO_LINT : BOOL
VAR_INPUT
	in : TOD;
	out : REFERENCE TO LINT;
END_VAR

out := TOD_TO_LINT(in);
TryConvert_TOD_TO_LINT := TRUE;

END_FUNCTION

// mobject-converters/Converters/TOD_TO_/TryConvert_TOD_TO_USINT
FUNCTION TryConvert_TOD_TO_USINT : BOOL
VAR_INPUT
	in : TOD;
	out : REFERENCE TO USINT;
END_VAR

IF in > DatatypeLimits.MAX_VALUE_OF_TOD_WHICH_CAN_BE_HELD_IN_A_USINT THEN
	RETURN;
END_IF

out := TOD_TO_USINT(in);
TryConvert_TOD_TO_USINT := TRUE;

END_FUNCTION

// mobject-converters/Converters/TOD_TO_/TryConvert_TOD_TO_UINT
FUNCTION TryConvert_TOD_TO_UINT : BOOL
VAR_INPUT
	in : TOD;
	out : REFERENCE TO UINT;
END_VAR

IF in > DatatypeLimits.MAX_VALUE_OF_TOD_WHICH_CAN_BE_HELD_IN_A_UINT THEN
	RETURN;
END_IF

out := TOD_TO_UINT(in);
TryConvert_TOD_TO_UINT := TRUE;

END_FUNCTION

// mobject-converters/Converters/TOD_TO_/TryConvert_TOD_TO_UDINT
FUNCTION TryConvert_TOD_TO_UDINT : BOOL
VAR_INPUT
	in : TOD;
	out : REFERENCE TO UDINT;
END_VAR

out := TOD_TO_UDINT(in);
TryConvert_TOD_TO_UDINT := TRUE;

END_FUNCTION

// mobject-converters/Converters/TOD_TO_/TryConvert_TOD_TO_ULINT
FUNCTION TryConvert_TOD_TO_ULINT : BOOL
VAR_INPUT
	in : TOD;
	out : REFERENCE TO ULINT;
END_VAR

out := TOD_TO_ULINT(in);
TryConvert_TOD_TO_ULINT := TRUE;

END_FUNCTION

// mobject-converters/Converters/TOD_TO_/TryConvert_TOD_TO_REAL
FUNCTION TryConvert_TOD_TO_REAL : BOOL
VAR_INPUT
	in : TOD;
	out : REFERENCE TO REAL;
END_VAR

out := TOD_TO_REAL(in);
TryConvert_TOD_TO_REAL := TRUE;

END_FUNCTION

// mobject-converters/Converters/TOD_TO_/TryConvert_TOD_TO_LREAL
FUNCTION TryConvert_TOD_TO_LREAL : BOOL
VAR_INPUT
	in : TOD;
	out : REFERENCE TO LREAL;
END_VAR

out := TOD_TO_LREAL(in);
TryConvert_TOD_TO_LREAL := TRUE;

END_FUNCTION

// mobject-converters/Converters/TOD_TO_/TryConvert_TOD_TO_TIME
FUNCTION TryConvert_TOD_TO_TIME : BOOL
VAR_INPUT
	in : TOD;
	out : REFERENCE TO TIME;
END_VAR

out := TOD_TO_TIME(in);
TryConvert_TOD_TO_TIME := TRUE;

END_FUNCTION

// mobject-converters/Converters/TOD_TO_/TryConvert_TOD_TO_TOD
FUNCTION TryConvert_TOD_TO_TOD : BOOL
VAR_INPUT
	in : TOD;
	out : REFERENCE TO TOD;
END_VAR

out := in;
TryConvert_TOD_TO_TOD := TRUE;

END_FUNCTION

// mobject-converters/Converters/TOD_TO_/TryConvert_TOD_TO_DATE
FUNCTION TryConvert_TOD_TO_DATE : BOOL
VAR_INPUT
	in : TOD;
	out : REFERENCE TO DATE;
END_VAR

out := TOD_TO_DATE(in);
TryConvert_TOD_TO_DATE := TRUE;

END_FUNCTION

// mobject-converters/Converters/TOD_TO_/TryConvert_TOD_TO_DT
FUNCTION TryConvert_TOD_TO_DT : BOOL
VAR_INPUT
	in : TOD;
	out : REFERENCE TO DT;
END_VAR

out := TOD_TO_DT(in);
TryConvert_TOD_TO_DT := TRUE;

END_FUNCTION

// mobject-datatypes/Primitive/_DT
{attribute 'linkalways'} 
{attribute 'no_explicit_call' := 'This FB is a CLASS and must be accessed using methods or properties'}
{attribute 'enable_dynamic_creation'}
FUNCTION_BLOCK _DT EXTENDS DatatypeBase implements I_DT
VAR
	localData : DT;
	activeData : REFERENCE TO DT REF= localData;
END_VAR

METHOD FB_init : BOOL
VAR_INPUT
	bInitRetains : BOOL; // if TRUE, the retain variables are initialized (warm start / cold start)
	bInCopyCode : BOOL;  // if TRUE, the instance afterwards gets moved WORDo the copy code (online change)
	InitialValue : DT;
END_VAR
localData := InitialValue;
END_METHOD

PROPERTY PUBLIC Address : PVOID
GET
Address := ADR(activeData);
END_GET
END_PROPERTY

METHOD PUBLIC ClearReference
VAR_INPUT
END_VAR
activeData REF= localData;
END_METHOD

METHOD PUBLIC Clone : I_Datatype
VAR
    pClone : POINTER TO _DT;
END_VAR
pClone := __NEW(_DT(InitialValue := Value));
Clone := pClone^;
END_METHOD

METHOD PUBLIC MakeReferenceTo
VAR_INPUT
	ReferenceTarget : REFERENCE TO DT;
END_VAR
activeData REF= ReferenceTarget;
END_METHOD

METHOD PUBLIC SerializeWith
VAR_INPUT
	Serializer : I_Serializer;
END_VAR
Serializer.AddDateTime(activeData);
END_METHOD

PROPERTY PUBLIC Size : UDINT
GET
Size := SIZEOF(activeData);
END_GET
END_PROPERTY

METHOD PUBLIC TryConvertTo : BOOL
VAR_INPUT
	Destination : ANY;
END_VAR
TryConvertTo := TryConvert_DT_To_Destination(activeData, Destination);
END_METHOD

METHOD PUBLIC TryConvertTo_ : BOOL
VAR_INPUT
	Destination : I_Datatype;
END_VAR
VAR
	resultofBitConversion : BOOL;
	destinationAs_BIT : I_BIT;
	destinationAs_BOOL : I_BOOL;
	destinationAs_BYTE : I_BYTE;
	destinationAs_DINT : I_DINT;
	destinationAs_DT : I_DT;
	destinationAs_DWORD : I_DWORD;
	destinationAs_INT : I_INT;
	destinationAs_LINT : I_LINT;
	destinationAs_LREAL : I_LREAL;
	destinationAs_LWORD : I_LWORD;
	destinationAs_REAL : I_REAL;
	destinationAs_SINT : I_SINT;
	destinationAs_STRING : I_STRING;
	destinationAs_TOD : I_TOD;
	destinationAs_UDINT : I_UDINT;
	destinationAs_UINT : I_UINT;
	destinationAs_ULINT : I_ULINT;
	destinationAs_USINT : I_USINT;
	destinationAs_WORD : I_WORD;
END_VAR
IF destination.TryResolveAs_BIT(destinationAs_BIT) AND_THEN TryConvert_DT_TO_BOOL(activeData, resultofBitConversion) THEN
	destinationAs_BIT.Value := resultOfBitConversion;
	TryConvertTo_ := TRUE;
	RETURN;
END_IF

IF destination.TryResolveAs_BOOL(destinationAs_BOOL) THEN
	TryConvertTo_ := TryConvert_DT_TO_BOOL(activeData, destinationAs_BOOL.Value);
	RETURN;
END_IF
		
IF destination.TryResolveAs_BYTE(destinationAs_BYTE) THEN
	TryConvertTo_ := TryConvert_DT_TO_BYTE(activeData, destinationAs_BYTE.Value);
	RETURN;
END_IF

IF destination.TryResolveAs_DINT(destinationAs_DINT) THEN
	TryConvertTo_ := TryConvert_DT_TO_DINT(activeData, destinationAs_DINT.Value);
	RETURN;
END_IF

IF destination.TryResolveAs_DT(destinationAs_DT) THEN
	TryConvertTo_ := TryConvert_DT_TO_DT(activeData, destinationAs_DT.Value);
	RETURN;
END_IF

IF destination.TryResolveAs_DWORD(destinationAs_DWORD) THEN
	TryConvertTo_ := TryConvert_DT_TO_DWORD(activeData, destinationAs_DWORD.Value);
	RETURN;
END_IF

IF destination.TryResolveAs_INT(destinationAs_INT) THEN
	TryConvertTo_ := TryConvert_DT_TO_INT(activeData, destinationAs_INT.Value);
	RETURN;
END_IF

IF destination.TryResolveAs_LINT(destinationAs_LINT) THEN
	TryConvertTo_ := TryConvert_DT_TO_LINT(activeData, destinationAs_LINT.Value);
	RETURN;
END_IF

IF destination.TryResolveAs_LREAL(destinationAs_LREAL) THEN
	TryConvertTo_ := TryConvert_DT_TO_LREAL(activeData, destinationAs_LREAL.Value);
	RETURN;
END_IF

IF destination.TryResolveAs_LWORD(destinationAs_LWORD) THEN
	TryConvertTo_ := TryConvert_DT_TO_LWORD(activeData, destinationAs_LWORD.Value);
	RETURN;
END_IF

IF destination.TryResolveAs_REAL(destinationAs_REAL) THEN
	TryConvertTo_ := TryConvert_DT_TO_REAL(activeData, destinationAs_REAL.Value);
	RETURN;
END_IF

IF destination.TryResolveAs_SINT(destinationAs_SINT) THEN
	TryConvertTo_ := TryConvert_DT_TO_SINT(activeData, destinationAs_SINT.Value);
	RETURN;
END_IF

IF destination.TryResolveAs_STRING(destinationAs_STRING) THEN
	TryConvertTo_ := TryConvert_DT_TO_STRING(activeData, destinationAs_STRING.Value);
	RETURN;
END_IF

IF destination.TryResolveAs_TOD(destinationAs_TOD) THEN
	TryConvertTo_ := TryConvert_DT_TO_TOD(activeData, destinationAs_TOD.Value);
	RETURN;
END_IF

IF destination.TryResolveAs_UDINT(destinationAs_UDINT) THEN
	TryConvertTo_ := TryConvert_DT_TO_UDINT(activeData, destinationAs_UDINT.Value);
	RETURN;
END_IF

IF destination.TryResolveAs_UINT(destinationAs_UINT) THEN
	TryConvertTo_ := TryConvert_DT_TO_UINT(activeData, destinationAs_UINT.Value);
	RETURN;
END_IF

IF destination.TryResolveAs_ULINT(destinationAs_ULINT) THEN
	TryConvertTo_ := TryConvert_DT_TO_ULINT(activeData, destinationAs_ULINT.Value);
	RETURN;
END_IF

IF destination.TryResolveAs_USINT(destinationAs_USINT) THEN
	TryConvertTo_ := TryConvert_DT_TO_USINT(activeData, destinationAs_USINT.Value);
	RETURN;
END_IF

IF destination.TryResolveAs_WORD(destinationAs_WORD) THEN
	TryConvertTo_ := TryConvert_DT_TO_WORD(activeData, destinationAs_WORD.Value);
	RETURN;
END_IF
END_METHOD

METHOD TryDeserializeFrom : BOOL
VAR_INPUT
	Deserializer : I_Deserializer;
	Feedback : I_DeserializerFeedback;
END_VAR
TryDeserializeFrom := Deserializer.TryGetDateTime(activeData, Feedback);
END_METHOD

METHOD TryMakeReferenceTo : BOOL
VAR_INPUT
	Target : I_Datatype;
END_VAR
VAR
	pTargetData : POINTER TO DT;
END_VAR
IF NOT IsEquivalentTo(Target) THEN
	RETURN;
END_IF

pTargetData := Target.Address;
activeData REF= pTargetData^;
TryMakeReferenceTo := TRUE;
END_METHOD

METHOD PUBLIC TryResolveAs_DT : BOOL
VAR_INPUT
	Destination : REFERENCE TO I_DT;
END_VAR
Destination := THIS^;
TryResolveAs_DT := TRUE;
END_METHOD

PROPERTY PUBLIC TypeName : T_MAXSTRING
GET
TypeName := 'DT';
END_GET
END_PROPERTY

{warning disable C5410}
PROPERTY PUBLIC Value : REFERENCE TO DT
{warning restore C5410}
GET
Value REF= activeData;
END_GET
END_PROPERTY

END_FUNCTION_BLOCK

// mobject-converters/Converters/DT_TO_/TryConvert_DT_TO_Destination
FUNCTION TryConvert_DT_TO_Destination : BOOL
VAR_INPUT
	in : DT;
	out : ANY;
END_VAR
VAR
	convertResult : BOOL := FALSE;
	convertAddress : PVOID;
	_BOOL : BOOL;
	_BYTE : BYTE;
	_WORD : WORD;
	_DWORD : DWORD;
	_LWORD : LWORD;
	_SINT : SINT;
	_INT : INT;
	_DINT : DINT;
	_LINT : LINT;
	_USINT : USINT;
	_UINT : UINT;
	_UDINT : UDINT;
	_ULINT : ULINT;
	_REAL : REAL;
	_LREAL : LREAL;
	_TIME : TIME;
	_TOD : TOD;
	_DATE : DATE;
	_DT : DT;
	_STRING : STRING;
END_VAR

CASE out.TypeClass OF
	__SYSTEM.TYPE_CLASS.TYPE_BOOL:
	
	convertResult := TryConvert_DT_TO_BOOL(in, _BOOL);
	IF convertResult THEN
		convertAddress := ADR(_BOOL);
	END_IF
	
	__SYSTEM.TYPE_CLASS.TYPE_BYTE:
	
	convertResult := TryConvert_DT_TO_BYTE(in, _BYTE);
	IF convertResult THEN
		convertAddress := ADR(_BYTE);
	END_IF
	
	__SYSTEM.TYPE_CLASS.TYPE_WORD:
	
	convertResult := TryConvert_DT_TO_WORD(in, _WORD);
	IF convertResult THEN
		convertAddress := ADR(_WORD);
	END_IF
	
	__SYSTEM.TYPE_CLASS.TYPE_DWORD:
	
	convertResult := TryConvert_DT_TO_DWORD(in, _DWORD);
	IF convertResult THEN
		convertAddress := ADR(_DWORD);
	END_IF
	
	__SYSTEM.TYPE_CLASS.TYPE_LWORD:
	
	convertResult := TryConvert_DT_TO_LWORD(in, _LWORD);
	IF convertResult THEN
		convertAddress := ADR(_LWORD);
	END_IF
	
	__SYSTEM.TYPE_CLASS.TYPE_SINT:
	
	convertResult := TryConvert_DT_TO_SINT(in, _SINT);
	IF convertResult THEN
		convertAddress := ADR(_SINT);
	END_IF
	
	__SYSTEM.TYPE_CLASS.TYPE_INT:
	
	convertResult := TryConvert_DT_TO_INT(in, _INT);
	IF convertResult THEN
		convertAddress := ADR(_INT);
	END_IF
	
	__SYSTEM.TYPE_CLASS.TYPE_DINT:
	
	convertResult := TryConvert_DT_TO_DINT(in, _DINT);
	IF convertResult THEN
		convertAddress := ADR(_DINT);
	END_IF
	
	__SYSTEM.TYPE_CLASS.TYPE_LINT:
	
	convertResult := TryConvert_DT_TO_LINT(in, _LINT);
	IF convertResult THEN
		convertAddress := ADR(_LINT);
	END_IF
	
	__SYSTEM.TYPE_CLASS.TYPE_USINT:
	
	convertResult := TryConvert_DT_TO_USINT(in, _USINT);
	IF convertResult THEN
		convertAddress := ADR(_USINT);
	END_IF
	
	__SYSTEM.TYPE_CLASS.TYPE_UINT:
	
	convertResult := TryConvert_DT_TO_UINT(in, _UINT);
	IF convertResult THEN
		convertAddress := ADR(_UINT);
	END_IF
	
	__SYSTEM.TYPE_CLASS.TYPE_UDINT:
	
	convertResult := TryConvert_DT_TO_UDINT(in, _UDINT);
	IF convertResult THEN
		convertAddress := ADR(_UDINT);
	END_IF
	
	__SYSTEM.TYPE_CLASS.TYPE_ULINT:
	
	convertResult := TryConvert_DT_TO_ULINT(in, _ULINT);
	IF convertResult THEN
		convertAddress := ADR(_ULINT);
	END_IF
	
	__SYSTEM.TYPE_CLASS.TYPE_REAL:
	
	convertResult := TryConvert_DT_TO_REAL(in, _REAL);
	IF convertResult THEN
		convertAddress := ADR(_REAL);
	END_IF
	
	__SYSTEM.TYPE_CLASS.TYPE_LREAL:
	
	convertResult := TryConvert_DT_TO_LREAL(in, _LREAL);
	IF convertResult THEN
		convertAddress := ADR(_LREAL);
	END_IF
	
	__SYSTEM.TYPE_CLASS.TYPE_TIME:
	
	convertResult := TryConvert_DT_TO_TIME(in, _TIME);
	IF convertResult THEN
		convertAddress := ADR(_TIME);
	END_IF
	
	__SYSTEM.TYPE_CLASS.TYPE_TIMEOFDAY:
	
	convertResult := TryConvert_DT_TO_TOD(in, _TOD);
	IF convertResult THEN
		convertAddress := ADR(_TOD);
	END_IF
	
	__SYSTEM.TYPE_CLASS.TYPE_DATE:
	
	convertResult := TryConvert_DT_TO_DATE(in, _DATE);
	IF convertResult THEN
		convertAddress := ADR(_DATE);
	END_IF
	
	__SYSTEM.TYPE_CLASS.TYPE_DATEANDTIME:
	
	convertResult := TryConvert_DT_TO_DT(in, _DT);
	IF convertResult THEN
		convertAddress := ADR(_DT);
	END_IF
	
	__SYSTEM.TYPE_CLASS.TYPE_STRING:
	
	convertResult := TryConvert_DT_TO_STRING(in, _STRING);
	IF convertResult THEN
		convertAddress := ADR(_STRING);
	END_IF
	
END_CASE

IF convertResult THEN
	memcpy(out.pValue,convertAddress,DINT_TO_UDINT(out.diSize));
END_IF

TryConvert_DT_TO_Destination := convertResult;

END_FUNCTION

// mobject-converters/Converters/DT_TO_/TryConvert_DT_TO_BOOL
FUNCTION TryConvert_DT_TO_BOOL : BOOL
VAR_INPUT
	in : DT;
	out : REFERENCE TO BOOL;
END_VAR

out := DT_TO_BOOL(in);
TryConvert_DT_TO_BOOL := TRUE;

END_FUNCTION

// mobject-converters/Converters/DT_TO_/TryConvert_DT_TO_BYTE
FUNCTION TryConvert_DT_TO_BYTE : BOOL
VAR_INPUT
	in : DT;
	out : REFERENCE TO BYTE;
END_VAR

IF in > DatatypeLimits.MAX_VALUE_OF_DT_WHICH_CAN_BE_HELD_IN_A_BYTE THEN
	RETURN;
END_IF

out := DT_TO_BYTE(in);
TryConvert_DT_TO_BYTE := TRUE;

END_FUNCTION

// mobject-converters/Converters/DT_TO_/TryConvert_DT_TO_WORD
FUNCTION TryConvert_DT_TO_WORD : BOOL
VAR_INPUT
	in : DT;
	out : REFERENCE TO WORD;
END_VAR

IF in > DatatypeLimits.MAX_VALUE_OF_DT_WHICH_CAN_BE_HELD_IN_A_WORD THEN
	RETURN;
END_IF

out := DT_TO_WORD(in);
TryConvert_DT_TO_WORD := TRUE;

END_FUNCTION

// mobject-converters/Converters/DT_TO_/TryConvert_DT_TO_DWORD
FUNCTION TryConvert_DT_TO_DWORD : BOOL
VAR_INPUT
	in : DT;
	out : REFERENCE TO DWORD;
END_VAR

out := DT_TO_DWORD(in);
TryConvert_DT_TO_DWORD := TRUE;

END_FUNCTION

// mobject-converters/Converters/DT_TO_/TryConvert_DT_TO_LWORD
FUNCTION TryConvert_DT_TO_LWORD : BOOL
VAR_INPUT
	in : DT;
	out : REFERENCE TO LWORD;
END_VAR

out := DT_TO_LWORD(in);
TryConvert_DT_TO_LWORD := TRUE;

END_FUNCTION

// mobject-converters/Converters/DT_TO_/TryConvert_DT_TO_SINT
FUNCTION TryConvert_DT_TO_SINT : BOOL
VAR_INPUT
	in : DT;
	out : REFERENCE TO SINT;
END_VAR

IF in > DatatypeLimits.MAX_VALUE_OF_DT_WHICH_CAN_BE_HELD_IN_A_SINT THEN
	RETURN;
END_IF

out := DT_TO_SINT(in);
TryConvert_DT_TO_SINT := TRUE;

END_FUNCTION

// mobject-converters/Converters/DT_TO_/TryConvert_DT_TO_INT
FUNCTION TryConvert_DT_TO_INT : BOOL
VAR_INPUT
	in : DT;
	out : REFERENCE TO INT;
END_VAR

IF in > DatatypeLimits.MAX_VALUE_OF_DT_WHICH_CAN_BE_HELD_IN_A_INT THEN
	RETURN;
END_IF

out := DT_TO_INT(in);
TryConvert_DT_TO_INT := TRUE;

END_FUNCTION

// mobject-converters/Converters/DT_TO_/TryConvert_DT_TO_DINT
FUNCTION TryConvert_DT_TO_DINT : BOOL
VAR_INPUT
	in : DT;
	out : REFERENCE TO DINT;
END_VAR

IF in > DatatypeLimits.MAX_VALUE_OF_DT_WHICH_CAN_BE_HELD_IN_A_DINT THEN
	RETURN;
END_IF

out := DT_TO_DINT(in);
TryConvert_DT_TO_DINT := TRUE;

END_FUNCTION

// mobject-converters/Converters/DT_TO_/TryConvert_DT_TO_LINT
FUNCTION TryConvert_DT_TO_LINT : BOOL
VAR_INPUT
	in : DT;
	out : REFERENCE TO LINT;
END_VAR

out := DT_TO_LINT(in);
TryConvert_DT_TO_LINT := TRUE;

END_FUNCTION

// mobject-converters/Converters/DT_TO_/TryConvert_DT_TO_USINT
FUNCTION TryConvert_DT_TO_USINT : BOOL
VAR_INPUT
	in : DT;
	out : REFERENCE TO USINT;
END_VAR

IF in > DatatypeLimits.MAX_VALUE_OF_DT_WHICH_CAN_BE_HELD_IN_A_USINT THEN
	RETURN;
END_IF

out := DT_TO_USINT(in);
TryConvert_DT_TO_USINT := TRUE;

END_FUNCTION

// mobject-converters/Converters/DT_TO_/TryConvert_DT_TO_UINT
FUNCTION TryConvert_DT_TO_UINT : BOOL
VAR_INPUT
	in : DT;
	out : REFERENCE TO UINT;
END_VAR

IF in > DatatypeLimits.MAX_VALUE_OF_DT_WHICH_CAN_BE_HELD_IN_A_UINT THEN
	RETURN;
END_IF

out := DT_TO_UINT(in);
TryConvert_DT_TO_UINT := TRUE;

END_FUNCTION

// mobject-converters/Converters/DT_TO_/TryConvert_DT_TO_UDINT
FUNCTION TryConvert_DT_TO_UDINT : BOOL
VAR_INPUT
	in : DT;
	out : REFERENCE TO UDINT;
END_VAR

out := DT_TO_UDINT(in);
TryConvert_DT_TO_UDINT := TRUE;

END_FUNCTION

// mobject-converters/Converters/DT_TO_/TryConvert_DT_TO_ULINT
FUNCTION TryConvert_DT_TO_ULINT : BOOL
VAR_INPUT
	in : DT;
	out : REFERENCE TO ULINT;
END_VAR

out := DT_TO_ULINT(in);
TryConvert_DT_TO_ULINT := TRUE;

END_FUNCTION

// mobject-converters/Converters/DT_TO_/TryConvert_DT_TO_REAL
FUNCTION TryConvert_DT_TO_REAL : BOOL
VAR_INPUT
	in : DT;
	out : REFERENCE TO REAL;
END_VAR

out := DT_TO_REAL(in);
TryConvert_DT_TO_REAL := TRUE;

END_FUNCTION

// mobject-converters/Converters/DT_TO_/TryConvert_DT_TO_LREAL
FUNCTION TryConvert_DT_TO_LREAL : BOOL
VAR_INPUT
	in : DT;
	out : REFERENCE TO LREAL;
END_VAR

out := DT_TO_LREAL(in);
TryConvert_DT_TO_LREAL := TRUE;

END_FUNCTION

// mobject-converters/Converters/DT_TO_/TryConvert_DT_TO_TIME
FUNCTION TryConvert_DT_TO_TIME : BOOL
VAR_INPUT
	in : DT;
	out : REFERENCE TO TIME;
END_VAR

IF in > DatatypeLimits.MAX_VALUE_OF_DT_WHICH_CAN_BE_HELD_IN_A_TIME THEN
	RETURN;
END_IF

out := DT_TO_TIME(in);
TryConvert_DT_TO_TIME := TRUE;

END_FUNCTION

// mobject-converters/Converters/DT_TO_/TryConvert_DT_TO_TOD
FUNCTION TryConvert_DT_TO_TOD : BOOL
VAR_INPUT
	in : DT;
	out : REFERENCE TO TOD;
END_VAR

IF in > DatatypeLimits.MAX_VALUE_OF_DT_WHICH_CAN_BE_HELD_IN_A_TOD THEN
	RETURN;
END_IF

out := DT_TO_TOD(in);
TryConvert_DT_TO_TOD := TRUE;

END_FUNCTION

// mobject-converters/Converters/DT_TO_/TryConvert_DT_TO_DATE
FUNCTION TryConvert_DT_TO_DATE : BOOL
VAR_INPUT
	in : DT;
	out : REFERENCE TO DATE;
END_VAR

out := DT_TO_DATE(in);
TryConvert_DT_TO_DATE := TRUE;

END_FUNCTION

// mobject-converters/Converters/DT_TO_/TryConvert_DT_TO_DT
FUNCTION TryConvert_DT_TO_DT : BOOL
VAR_INPUT
	in : DT;
	out : REFERENCE TO DT;
END_VAR

out := in;
TryConvert_DT_TO_DT := TRUE;

END_FUNCTION

// mobject-converters/Converters/DT_TO_/TryConvert_DT_TO_STRING
FUNCTION TryConvert_DT_TO_STRING : BOOL
VAR_INPUT
	in : DT;
	out : REFERENCE TO STRING;
END_VAR

out := DT_TO_STRING(in);
TryConvert_DT_TO_STRING := TRUE;

END_FUNCTION

// mobject-datatypes/Primitive/_STRING
{attribute 'linkalways'} 
{attribute 'no_explicit_call' := 'This FB is a CLASS and must be accessed using methods or properties'}
{attribute 'enable_dynamic_creation'}
FUNCTION_BLOCK _STRING EXTENDS DatatypeBase implements I_STRING
VAR
	localData : T_MaxString;
	activeData : REFERENCE TO T_MaxString REF= localData;
END_VAR

METHOD FB_init : BOOL
VAR_INPUT
	bInitRetains : BOOL; // if TRUE, the retain variables are initialized (warm start / cold start)
	bInCopyCode : BOOL;  // if TRUE, the instance afterwards gets moved WORDo the copy code (online change)
	InitialValue : T_MaxString;
END_VAR
localData := InitialValue;
END_METHOD

PROPERTY PUBLIC Address : PVOID
GET
Address := ADR(activeData);
END_GET
END_PROPERTY

METHOD PUBLIC ClearReference
VAR_INPUT
END_VAR
activeData REF= localData;
END_METHOD

METHOD PUBLIC Clone : I_Datatype
VAR
    pClone : POINTER TO _STRING;
END_VAR
pClone := __NEW(_STRING(InitialValue := Value));
Clone := pClone^;
END_METHOD

PROPERTY PUBLIC Length : INT
GET
Length := len(activeData);
END_GET
END_PROPERTY

METHOD PUBLIC MakeReferenceTo
VAR_INPUT
	ReferenceTarget : REFERENCE TO T_MaxString;
END_VAR
activeData REF= ReferenceTarget;
END_METHOD

METHOD PUBLIC SerializeWith
VAR_INPUT
	Serializer : I_Serializer;
END_VAR
Serializer.AddString(activeData);
END_METHOD

PROPERTY PUBLIC Size : UDINT
GET
Size := SIZEOF(activeData);
END_GET
END_PROPERTY

METHOD PUBLIC TryConvertTo : BOOL
VAR_INPUT
	Destination : ANY;
END_VAR
TryConvertTo := TryConvert_STRING_TO_Destination(activeData, Destination);
END_METHOD

METHOD PUBLIC TryConvertTo_ : BOOL
VAR_INPUT
	Destination : I_Datatype;
END_VAR
VAR
	resultofBitConversion : BOOL;
	destinationAs_BIT : I_BIT;
	destinationAs_BOOL : I_BOOL;
	destinationAs_BYTE : I_BYTE;
	destinationAs_DINT : I_DINT;
	destinationAs_DT : I_DT;
	destinationAs_DWORD : I_DWORD;
	destinationAs_INT : I_INT;
	destinationAs_LINT : I_LINT;
	destinationAs_LREAL : I_LREAL;
	destinationAs_LWORD : I_LWORD;
	destinationAs_REAL : I_REAL;
	destinationAs_SINT : I_SINT;
	destinationAs_STRING : I_STRING;
	destinationAs_TOD : I_TOD;
	destinationAs_UDINT : I_UDINT;
	destinationAs_UINT : I_UINT;
	destinationAs_ULINT : I_ULINT;
	destinationAs_USINT : I_USINT;
	destinationAs_WORD : I_WORD;
END_VAR
IF destination.TryResolveAs_BIT(destinationAs_BIT) AND_THEN TryConvert_STRING_TO_BOOL(activeData, resultofBitConversion) THEN
	destinationAs_BIT.Value := resultOfBitConversion;
	TryConvertTo_ := TRUE;
	RETURN;
END_IF

IF destination.TryResolveAs_BOOL(destinationAs_BOOL) THEN
	TryConvertTo_ := TryConvert_STRING_TO_BOOL(activeData, destinationAs_BOOL.Value);
	RETURN;
END_IF
		
IF destination.TryResolveAs_BYTE(destinationAs_BYTE) THEN
	TryConvertTo_ := TryConvert_STRING_TO_BYTE(activeData, destinationAs_BYTE.Value);
	RETURN;
END_IF

IF destination.TryResolveAs_DINT(destinationAs_DINT) THEN
	TryConvertTo_ := TryConvert_STRING_TO_DINT(activeData, destinationAs_DINT.Value);
	RETURN;
END_IF

IF destination.TryResolveAs_DT(destinationAs_DT) THEN
	TryConvertTo_ := TryConvert_STRING_TO_DT(activeData, destinationAs_DT.Value);
	RETURN;
END_IF

IF destination.TryResolveAs_DWORD(destinationAs_DWORD) THEN
	TryConvertTo_ := TryConvert_STRING_TO_DWORD(activeData, destinationAs_DWORD.Value);
	RETURN;
END_IF

IF destination.TryResolveAs_INT(destinationAs_INT) THEN
	TryConvertTo_ := TryConvert_STRING_TO_INT(activeData, destinationAs_INT.Value);
	RETURN;
END_IF

IF destination.TryResolveAs_LINT(destinationAs_LINT) THEN
	TryConvertTo_ := TryConvert_STRING_TO_LINT(activeData, destinationAs_LINT.Value);
	RETURN;
END_IF

IF destination.TryResolveAs_LREAL(destinationAs_LREAL) THEN
	TryConvertTo_ := TryConvert_STRING_TO_LREAL(activeData, destinationAs_LREAL.Value);
	RETURN;
END_IF

IF destination.TryResolveAs_LWORD(destinationAs_LWORD) THEN
	TryConvertTo_ := TryConvert_STRING_TO_LWORD(activeData, destinationAs_LWORD.Value);
	RETURN;
END_IF

IF destination.TryResolveAs_REAL(destinationAs_REAL) THEN
	TryConvertTo_ := TryConvert_STRING_TO_REAL(activeData, destinationAs_REAL.Value);
	RETURN;
END_IF

IF destination.TryResolveAs_SINT(destinationAs_SINT) THEN
	TryConvertTo_ := TryConvert_STRING_TO_SINT(activeData, destinationAs_SINT.Value);
	RETURN;
END_IF

IF destination.TryResolveAs_STRING(destinationAs_STRING) THEN
	TryConvertTo_ := TryConvert_STRING_TO_STRING(activeData, destinationAs_STRING.Value);
	RETURN;
END_IF

IF destination.TryResolveAs_TOD(destinationAs_TOD) THEN
	TryConvertTo_ := TryConvert_STRING_TO_TOD(activeData, destinationAs_TOD.Value);
	RETURN;
END_IF

IF destination.TryResolveAs_UDINT(destinationAs_UDINT) THEN
	TryConvertTo_ := TryConvert_STRING_TO_UDINT(activeData, destinationAs_UDINT.Value);
	RETURN;
END_IF

IF destination.TryResolveAs_UINT(destinationAs_UINT) THEN
	TryConvertTo_ := TryConvert_STRING_TO_UINT(activeData, destinationAs_UINT.Value);
	RETURN;
END_IF

IF destination.TryResolveAs_ULINT(destinationAs_ULINT) THEN
	TryConvertTo_ := TryConvert_STRING_TO_ULINT(activeData, destinationAs_ULINT.Value);
	RETURN;
END_IF

IF destination.TryResolveAs_USINT(destinationAs_USINT) THEN
	TryConvertTo_ := TryConvert_STRING_TO_USINT(activeData, destinationAs_USINT.Value);
	RETURN;
END_IF

IF destination.TryResolveAs_WORD(destinationAs_WORD) THEN
	TryConvertTo_ := TryConvert_STRING_TO_WORD(activeData, destinationAs_WORD.Value);
	RETURN;
END_IF
END_METHOD

METHOD TryDeserializeFrom : BOOL
VAR_INPUT
	Deserializer : I_Deserializer;
	Feedback : I_DeserializerFeedback;
END_VAR
TryDeserializeFrom := Deserializer.TryGetString(activeData, Feedback);
END_METHOD

METHOD TryMakeReferenceTo : BOOL
VAR_INPUT
	Target : I_Datatype;
END_VAR
VAR
	pTargetData : POINTER TO T_MaxString;
END_VAR
IF NOT IsEquivalentTo(Target) THEN
	RETURN;
END_IF

pTargetData := Target.Address;
activeData REF= pTargetData^;
TryMakeReferenceTo := TRUE;
END_METHOD

METHOD PUBLIC TryResolveAs_STRING : BOOL
VAR_INPUT
	Destination : REFERENCE TO I_STRING;
END_VAR
Destination := THIS^;
TryResolveAs_STRING := TRUE;
END_METHOD

PROPERTY PUBLIC TypeName : T_MAXSTRING
GET
TypeName := 'STRING';
END_GET
END_PROPERTY

{warning disable C5410}
PROPERTY PUBLIC Value : REFERENCE TO T_MaxString
{warning restore C5410}
GET
Value REF= activeData;
END_GET
END_PROPERTY

END_FUNCTION_BLOCK

// mobject-converters/Converters/STRING_TO_/TryConvert_STRING_TO_Destination
FUNCTION TryConvert_STRING_TO_Destination : BOOL
VAR_INPUT
	in : STRING;
	out : ANY;
END_VAR
VAR
	convertResult : BOOL := FALSE;
	convertAddress : PVOID;
	_BOOL : BOOL;
	_BYTE : BYTE;
	_WORD : WORD;
	_DWORD : DWORD;
	_LWORD : LWORD;
	_SINT : SINT;
	_INT : INT;
	_DINT : DINT;
	_LINT : LINT;
	_USINT : USINT;
	_UINT : UINT;
	_UDINT : UDINT;
	_ULINT : ULINT;
	_REAL : REAL;
	_LREAL : LREAL;
	_TIME : TIME;
	_TOD : TOD;
	_DATE : DATE;
	_DT : DT;
	_STRING : STRING;
END_VAR

CASE out.TypeClass OF
	__SYSTEM.TYPE_CLASS.TYPE_BOOL:
	
	convertResult := TryConvert_STRING_TO_BOOL(in, _BOOL);
	IF convertResult THEN
		convertAddress := ADR(_BOOL);
	END_IF
	
	__SYSTEM.TYPE_CLASS.TYPE_BYTE:
	
	convertResult := TryConvert_STRING_TO_BYTE(in, _BYTE);
	IF convertResult THEN
		convertAddress := ADR(_BYTE);
	END_IF
	
	__SYSTEM.TYPE_CLASS.TYPE_WORD:
	
	convertResult := TryConvert_STRING_TO_WORD(in, _WORD);
	IF convertResult THEN
		convertAddress := ADR(_WORD);
	END_IF
	
	__SYSTEM.TYPE_CLASS.TYPE_DWORD:
	
	convertResult := TryConvert_STRING_TO_DWORD(in, _DWORD);
	IF convertResult THEN
		convertAddress := ADR(_DWORD);
	END_IF
	
	__SYSTEM.TYPE_CLASS.TYPE_LWORD:
	
	convertResult := TryConvert_STRING_TO_LWORD(in, _LWORD);
	IF convertResult THEN
		convertAddress := ADR(_LWORD);
	END_IF
	
	__SYSTEM.TYPE_CLASS.TYPE_SINT:
	
	convertResult := TryConvert_STRING_TO_SINT(in, _SINT);
	IF convertResult THEN
		convertAddress := ADR(_SINT);
	END_IF
	
	__SYSTEM.TYPE_CLASS.TYPE_INT:
	
	convertResult := TryConvert_STRING_TO_INT(in, _INT);
	IF convertResult THEN
		convertAddress := ADR(_INT);
	END_IF
	
	__SYSTEM.TYPE_CLASS.TYPE_DINT:
	
	convertResult := TryConvert_STRING_TO_DINT(in, _DINT);
	IF convertResult THEN
		convertAddress := ADR(_DINT);
	END_IF
	
	__SYSTEM.TYPE_CLASS.TYPE_LINT:
	
	convertResult := TryConvert_STRING_TO_LINT(in, _LINT);
	IF convertResult THEN
		convertAddress := ADR(_LINT);
	END_IF
	
	__SYSTEM.TYPE_CLASS.TYPE_USINT:
	
	convertResult := TryConvert_STRING_TO_USINT(in, _USINT);
	IF convertResult THEN
		convertAddress := ADR(_USINT);
	END_IF
	
	__SYSTEM.TYPE_CLASS.TYPE_UINT:
	
	convertResult := TryConvert_STRING_TO_UINT(in, _UINT);
	IF convertResult THEN
		convertAddress := ADR(_UINT);
	END_IF
	
	__SYSTEM.TYPE_CLASS.TYPE_UDINT:
	
	convertResult := TryConvert_STRING_TO_UDINT(in, _UDINT);
	IF convertResult THEN
		convertAddress := ADR(_UDINT);
	END_IF
	
	__SYSTEM.TYPE_CLASS.TYPE_ULINT:
	
	convertResult := TryConvert_STRING_TO_ULINT(in, _ULINT);
	IF convertResult THEN
		convertAddress := ADR(_ULINT);
	END_IF
	
	__SYSTEM.TYPE_CLASS.TYPE_REAL:
	
	convertResult := TryConvert_STRING_TO_REAL(in, _REAL);
	IF convertResult THEN
		convertAddress := ADR(_REAL);
	END_IF
	
	__SYSTEM.TYPE_CLASS.TYPE_LREAL:
	
	convertResult := TryConvert_STRING_TO_LREAL(in, _LREAL);
	IF convertResult THEN
		convertAddress := ADR(_LREAL);
	END_IF
	
	__SYSTEM.TYPE_CLASS.TYPE_TIME:
	
	convertResult := TryConvert_STRING_TO_TIME(in, _TIME);
	IF convertResult THEN
		convertAddress := ADR(_TIME);
	END_IF
	
	__SYSTEM.TYPE_CLASS.TYPE_TIMEOFDAY:
	
	convertResult := TryConvert_STRING_TO_TOD(in, _TOD);
	IF convertResult THEN
		convertAddress := ADR(_TOD);
	END_IF
	
	__SYSTEM.TYPE_CLASS.TYPE_DATE:
	
	convertResult := TryConvert_STRING_TO_DATE(in, _DATE);
	IF convertResult THEN
		convertAddress := ADR(_DATE);
	END_IF
	
	__SYSTEM.TYPE_CLASS.TYPE_DATEANDTIME:
	
	convertResult := TryConvert_STRING_TO_DT(in, _DT);
	IF convertResult THEN
		convertAddress := ADR(_DT);
	END_IF
	
	__SYSTEM.TYPE_CLASS.TYPE_STRING:
	
	convertResult := TryConvert_STRING_TO_STRING(in, _STRING);
	IF convertResult THEN
		convertAddress := ADR(_STRING);
	END_IF
	
END_CASE

IF convertResult THEN
	memcpy(out.pValue,convertAddress,DINT_TO_UDINT(out.diSize));
END_IF

TryConvert_STRING_TO_Destination := convertResult;

END_FUNCTION

// mobject-converters/Converters/STRING_TO_/TryConvert_STRING_TO_BOOL
FUNCTION TryConvert_STRING_TO_BOOL : BOOL
VAR_INPUT
	in : STRING;
	out : REFERENCE TO BOOL;
END_VAR

out := STRING_TO_BOOL(in);
TryConvert_STRING_TO_BOOL := TRUE;

END_FUNCTION

// mobject-converters/Converters/STRING_TO_/TryConvert_STRING_TO_BYTE
FUNCTION TryConvert_STRING_TO_BYTE : BOOL
VAR_INPUT
	in : STRING;
	out : REFERENCE TO BYTE;
END_VAR

IF in <> BYTE_TO_STRING(STRING_TO_BYTE(in)) THEN
	RETURN;
END_IF

out := STRING_TO_BYTE(in);
TryConvert_STRING_TO_BYTE := TRUE;

END_FUNCTION

// mobject-converters/Converters/STRING_TO_/TryConvert_STRING_TO_WORD
FUNCTION TryConvert_STRING_TO_WORD : BOOL
VAR_INPUT
	in : STRING;
	out : REFERENCE TO WORD;
END_VAR

IF in <> WORD_TO_STRING(STRING_TO_WORD(in)) THEN
	RETURN;
END_IF

out := STRING_TO_WORD(in);
TryConvert_STRING_TO_WORD := TRUE;

END_FUNCTION

// mobject-converters/Converters/STRING_TO_/TryConvert_STRING_TO_DWORD
FUNCTION TryConvert_STRING_TO_DWORD : BOOL
VAR_INPUT
	in : STRING;
	out : REFERENCE TO DWORD;
END_VAR

IF in <> DWORD_TO_STRING(STRING_TO_DWORD(in)) THEN
	RETURN;
END_IF

out := STRING_TO_DWORD(in);
TryConvert_STRING_TO_DWORD := TRUE;

END_FUNCTION

// mobject-converters/Converters/STRING_TO_/TryConvert_STRING_TO_LWORD
FUNCTION TryConvert_STRING_TO_LWORD : BOOL
VAR_INPUT
	in : STRING;
	out : REFERENCE TO LWORD;
END_VAR

IF in <> LWORD_TO_STRING(STRING_TO_LWORD(in)) THEN
	RETURN;
END_IF

out := STRING_TO_LWORD(in);
TryConvert_STRING_TO_LWORD := TRUE;

END_FUNCTION

// mobject-converters/Converters/STRING_TO_/TryConvert_STRING_TO_SINT
FUNCTION TryConvert_STRING_TO_SINT : BOOL
VAR_INPUT
	in : STRING;
	out : REFERENCE TO SINT;
END_VAR

IF in <> SINT_TO_STRING(STRING_TO_SINT(in)) THEN
	RETURN;
END_IF

out := STRING_TO_SINT(in);
TryConvert_STRING_TO_SINT := TRUE;

END_FUNCTION

// mobject-converters/Converters/STRING_TO_/TryConvert_STRING_TO_INT
FUNCTION TryConvert_STRING_TO_INT : BOOL
VAR_INPUT
	in : STRING;
	out : REFERENCE TO INT;
END_VAR

IF in <> INT_TO_STRING(STRING_TO_INT(in)) THEN
	RETURN;
END_IF

out := STRING_TO_INT(in);
TryConvert_STRING_TO_INT := TRUE;

END_FUNCTION

// mobject-converters/Converters/STRING_TO_/TryConvert_STRING_TO_DINT
FUNCTION TryConvert_STRING_TO_DINT : BOOL
VAR_INPUT
	in : STRING;
	out : REFERENCE TO DINT;
END_VAR

IF in <> DINT_TO_STRING(STRING_TO_DINT(in)) THEN
	RETURN;
END_IF

out := STRING_TO_DINT(in);
TryConvert_STRING_TO_DINT := TRUE;

END_FUNCTION

// mobject-converters/Converters/STRING_TO_/TryConvert_STRING_TO_LINT
FUNCTION TryConvert_STRING_TO_LINT : BOOL
VAR_INPUT
	in : STRING;
	out : REFERENCE TO LINT;
END_VAR

IF in <> LINT_TO_STRING(STRING_TO_LINT(in)) THEN
	RETURN;
END_IF

out := STRING_TO_LINT(in);
TryConvert_STRING_TO_LINT := TRUE;

END_FUNCTION

// mobject-converters/Converters/STRING_TO_/TryConvert_STRING_TO_USINT
FUNCTION TryConvert_STRING_TO_USINT : BOOL
VAR_INPUT
	in : STRING;
	out : REFERENCE TO USINT;
END_VAR

IF in <> USINT_TO_STRING(STRING_TO_USINT(in)) THEN
	RETURN;
END_IF

out := STRING_TO_USINT(in);
TryConvert_STRING_TO_USINT := TRUE;

END_FUNCTION

// mobject-converters/Converters/STRING_TO_/TryConvert_STRING_TO_UINT
FUNCTION TryConvert_STRING_TO_UINT : BOOL
VAR_INPUT
	in : STRING;
	out : REFERENCE TO UINT;
END_VAR

IF in <> UINT_TO_STRING(STRING_TO_UINT(in)) THEN
	RETURN;
END_IF

out := STRING_TO_UINT(in);
TryConvert_STRING_TO_UINT := TRUE;

END_FUNCTION

// mobject-converters/Converters/STRING_TO_/TryConvert_STRING_TO_UDINT
FUNCTION TryConvert_STRING_TO_UDINT : BOOL
VAR_INPUT
	in : STRING;
	out : REFERENCE TO UDINT;
END_VAR

IF in <> UDINT_TO_STRING(STRING_TO_UDINT(in)) THEN
	RETURN;
END_IF

out := STRING_TO_UDINT(in);
TryConvert_STRING_TO_UDINT := TRUE;

END_FUNCTION

// mobject-converters/Converters/STRING_TO_/TryConvert_STRING_TO_ULINT
FUNCTION TryConvert_STRING_TO_ULINT : BOOL
VAR_INPUT
	in : STRING;
	out : REFERENCE TO ULINT;
END_VAR

IF in <> ULINT_TO_STRING(STRING_TO_ULINT(in)) THEN
	RETURN;
END_IF

out := STRING_TO_ULINT(in);
TryConvert_STRING_TO_ULINT := TRUE;

END_FUNCTION

// mobject-converters/Converters/STRING_TO_/TryConvert_STRING_TO_REAL
FUNCTION TryConvert_STRING_TO_REAL : BOOL
VAR_INPUT
	in : STRING;
	out : REFERENCE TO REAL;
END_VAR

IF in <> REAL_TO_STRING(STRING_TO_REAL(in)) THEN
	RETURN;
END_IF

out := STRING_TO_REAL(in);
TryConvert_STRING_TO_REAL := TRUE;

END_FUNCTION

// mobject-converters/Converters/STRING_TO_/TryConvert_STRING_TO_LREAL
FUNCTION TryConvert_STRING_TO_LREAL : BOOL
VAR_INPUT
	in : STRING;
	out : REFERENCE TO LREAL;
END_VAR

IF in <> LREAL_TO_STRING(STRING_TO_LREAL(in)) THEN
	RETURN;
END_IF

out := STRING_TO_LREAL(in);
TryConvert_STRING_TO_LREAL := TRUE;

END_FUNCTION

// mobject-converters/Converters/STRING_TO_/TryConvert_STRING_TO_TIME
FUNCTION TryConvert_STRING_TO_TIME : BOOL
VAR_INPUT
	in : STRING;
	out : REFERENCE TO TIME;
END_VAR

IF in <> TIME_TO_STRING(STRING_TO_TIME(in)) THEN
	RETURN;
END_IF

out := STRING_TO_TIME(in);
TryConvert_STRING_TO_TIME := TRUE;

END_FUNCTION

// mobject-converters/Converters/STRING_TO_/TryConvert_STRING_TO_TOD
FUNCTION TryConvert_STRING_TO_TOD : BOOL
VAR_INPUT
	in : STRING;
	out : REFERENCE TO TOD;
END_VAR

IF in <> TOD_TO_STRING(STRING_TO_TOD(in)) THEN
	RETURN;
END_IF

out := STRING_TO_TOD(in);
TryConvert_STRING_TO_TOD := TRUE;

END_FUNCTION

// mobject-converters/Converters/STRING_TO_/TryConvert_STRING_TO_DATE
FUNCTION TryConvert_STRING_TO_DATE : BOOL
VAR_INPUT
	in : STRING;
	out : REFERENCE TO DATE;
END_VAR

IF in <> DATE_TO_STRING(STRING_TO_DATE(in)) THEN
	RETURN;
END_IF

out := STRING_TO_DATE(in);
TryConvert_STRING_TO_DATE := TRUE;

END_FUNCTION

// mobject-converters/Converters/STRING_TO_/TryConvert_STRING_TO_DT
FUNCTION TryConvert_STRING_TO_DT : BOOL
VAR_INPUT
	in : STRING;
	out : REFERENCE TO DT;
END_VAR

IF in <> DT_TO_STRING(STRING_TO_DT(in)) THEN
	RETURN;
END_IF

out := STRING_TO_DT(in);
TryConvert_STRING_TO_DT := TRUE;

END_FUNCTION

// mobject-converters/Converters/STRING_TO_/TryConvert_STRING_TO_STRING
FUNCTION TryConvert_STRING_TO_STRING : BOOL
VAR_INPUT
	in : STRING;
	out : REFERENCE TO STRING;
END_VAR

out := in;
TryConvert_STRING_TO_STRING := TRUE;

END_FUNCTION

// mobject-converters/Converters/TOD_TO_/TryConvert_TOD_TO_STRING
FUNCTION TryConvert_TOD_TO_STRING : BOOL
VAR_INPUT
	in : TOD;
	out : REFERENCE TO STRING;
END_VAR

out := TOD_TO_STRING(in);
TryConvert_TOD_TO_STRING := TRUE;

END_FUNCTION

// mobject-converters/Converters/LREAL_TO_/TryConvert_LREAL_TO_DATE
FUNCTION TryConvert_LREAL_TO_DATE : BOOL
VAR_INPUT
	in : LREAL;
	out : REFERENCE TO DATE;
END_VAR

IF in > DatatypeLimits.MAX_VALUE_OF_LREAL_WHICH_CAN_BE_HELD_IN_A_DATE THEN
	RETURN;
END_IF

IF in < DatatypeLimits.MIN_VALUE_OF_LREAL_WHICH_CAN_BE_HELD_IN_A_DATE THEN
	RETURN;
END_IF

out := LREAL_TO_DATE(in);
TryConvert_LREAL_TO_DATE := TRUE;

END_FUNCTION

// mobject-converters/Converters/LREAL_TO_/TryConvert_LREAL_TO_DT
FUNCTION TryConvert_LREAL_TO_DT : BOOL
VAR_INPUT
	in : LREAL;
	out : REFERENCE TO DT;
END_VAR

IF in > DatatypeLimits.MAX_VALUE_OF_LREAL_WHICH_CAN_BE_HELD_IN_A_DT THEN
	RETURN;
END_IF

IF in < DatatypeLimits.MIN_VALUE_OF_LREAL_WHICH_CAN_BE_HELD_IN_A_DT THEN
	RETURN;
END_IF

out := LREAL_TO_DT(in);
TryConvert_LREAL_TO_DT := TRUE;

END_FUNCTION

// mobject-converters/Converters/LREAL_TO_/TryConvert_LREAL_TO_STRING
FUNCTION TryConvert_LREAL_TO_STRING : BOOL
VAR_INPUT
	in : LREAL;
	out : REFERENCE TO STRING;
END_VAR

IF in > DatatypeLimits.MAX_VALUE_OF_LREAL_WHICH_CAN_BE_HELD_IN_A_STRING THEN
	RETURN;
END_IF

IF in < DatatypeLimits.MIN_VALUE_OF_LREAL_WHICH_CAN_BE_HELD_IN_A_STRING THEN
	RETURN;
END_IF

out := LREAL_TO_STRING(in);
TryConvert_LREAL_TO_STRING := TRUE;

END_FUNCTION

// mobject-converters/Converters/REAL_TO_/TryConvert_REAL_TO_TIME
FUNCTION TryConvert_REAL_TO_TIME : BOOL
VAR_INPUT
	in : REAL;
	out : REFERENCE TO TIME;
END_VAR

IF in > DatatypeLimits.MAX_VALUE_OF_REAL_WHICH_CAN_BE_HELD_IN_A_TIME THEN
	RETURN;
END_IF

IF in < DatatypeLimits.MIN_VALUE_OF_REAL_WHICH_CAN_BE_HELD_IN_A_TIME THEN
	RETURN;
END_IF

out := REAL_TO_TIME(in);
TryConvert_REAL_TO_TIME := TRUE;

END_FUNCTION

// mobject-converters/Converters/REAL_TO_/TryConvert_REAL_TO_TOD
FUNCTION TryConvert_REAL_TO_TOD : BOOL
VAR_INPUT
	in : REAL;
	out : REFERENCE TO TOD;
END_VAR

IF in > DatatypeLimits.MAX_VALUE_OF_REAL_WHICH_CAN_BE_HELD_IN_A_TOD THEN
	RETURN;
END_IF

IF in < DatatypeLimits.MIN_VALUE_OF_REAL_WHICH_CAN_BE_HELD_IN_A_TOD THEN
	RETURN;
END_IF

out := REAL_TO_TOD(in);
TryConvert_REAL_TO_TOD := TRUE;

END_FUNCTION

// mobject-converters/Converters/REAL_TO_/TryConvert_REAL_TO_DATE
FUNCTION TryConvert_REAL_TO_DATE : BOOL
VAR_INPUT
	in : REAL;
	out : REFERENCE TO DATE;
END_VAR

IF in > DatatypeLimits.MAX_VALUE_OF_REAL_WHICH_CAN_BE_HELD_IN_A_DATE THEN
	RETURN;
END_IF

IF in < DatatypeLimits.MIN_VALUE_OF_REAL_WHICH_CAN_BE_HELD_IN_A_DATE THEN
	RETURN;
END_IF

out := REAL_TO_DATE(in);
TryConvert_REAL_TO_DATE := TRUE;

END_FUNCTION

// mobject-converters/Converters/REAL_TO_/TryConvert_REAL_TO_DT
FUNCTION TryConvert_REAL_TO_DT : BOOL
VAR_INPUT
	in : REAL;
	out : REFERENCE TO DT;
END_VAR

IF in > DatatypeLimits.MAX_VALUE_OF_REAL_WHICH_CAN_BE_HELD_IN_A_DT THEN
	RETURN;
END_IF

IF in < DatatypeLimits.MIN_VALUE_OF_REAL_WHICH_CAN_BE_HELD_IN_A_DT THEN
	RETURN;
END_IF

out := REAL_TO_DT(in);
TryConvert_REAL_TO_DT := TRUE;

END_FUNCTION

// mobject-converters/Converters/REAL_TO_/TryConvert_REAL_TO_STRING
FUNCTION TryConvert_REAL_TO_STRING : BOOL
VAR_INPUT
	in : REAL;
	out : REFERENCE TO STRING;
END_VAR

out := REAL_TO_STRING(in);
TryConvert_REAL_TO_STRING := TRUE;

END_FUNCTION

// mobject-converters/Converters/ULINT_TO_/TryConvert_ULINT_TO_LREAL
FUNCTION TryConvert_ULINT_TO_LREAL : BOOL
VAR_INPUT
	in : ULINT;
	out : REFERENCE TO LREAL;
END_VAR

out := ULINT_TO_LREAL(in);
TryConvert_ULINT_TO_LREAL := TRUE;

END_FUNCTION

// mobject-converters/Converters/ULINT_TO_/TryConvert_ULINT_TO_TIME
FUNCTION TryConvert_ULINT_TO_TIME : BOOL
VAR_INPUT
	in : ULINT;
	out : REFERENCE TO TIME;
END_VAR

IF in > DatatypeLimits.MAX_VALUE_OF_ULINT_WHICH_CAN_BE_HELD_IN_A_TIME THEN
	RETURN;
END_IF

out := ULINT_TO_TIME(in);
TryConvert_ULINT_TO_TIME := TRUE;

END_FUNCTION

// mobject-converters/Converters/ULINT_TO_/TryConvert_ULINT_TO_TOD
FUNCTION TryConvert_ULINT_TO_TOD : BOOL
VAR_INPUT
	in : ULINT;
	out : REFERENCE TO TOD;
END_VAR

IF in > DatatypeLimits.MAX_VALUE_OF_ULINT_WHICH_CAN_BE_HELD_IN_A_TOD THEN
	RETURN;
END_IF

out := ULINT_TO_TOD(in);
TryConvert_ULINT_TO_TOD := TRUE;

END_FUNCTION

// mobject-converters/Converters/ULINT_TO_/TryConvert_ULINT_TO_DATE
FUNCTION TryConvert_ULINT_TO_DATE : BOOL
VAR_INPUT
	in : ULINT;
	out : REFERENCE TO DATE;
END_VAR

IF in > DatatypeLimits.MAX_VALUE_OF_ULINT_WHICH_CAN_BE_HELD_IN_A_DATE THEN
	RETURN;
END_IF

out := ULINT_TO_DATE(in);
TryConvert_ULINT_TO_DATE := TRUE;

END_FUNCTION

// mobject-converters/Converters/ULINT_TO_/TryConvert_ULINT_TO_DT
FUNCTION TryConvert_ULINT_TO_DT : BOOL
VAR_INPUT
	in : ULINT;
	out : REFERENCE TO DT;
END_VAR

IF in > DatatypeLimits.MAX_VALUE_OF_ULINT_WHICH_CAN_BE_HELD_IN_A_DT THEN
	RETURN;
END_IF

out := ULINT_TO_DT(in);
TryConvert_ULINT_TO_DT := TRUE;

END_FUNCTION

// mobject-converters/Converters/ULINT_TO_/TryConvert_ULINT_TO_STRING
FUNCTION TryConvert_ULINT_TO_STRING : BOOL
VAR_INPUT
	in : ULINT;
	out : REFERENCE TO STRING;
END_VAR

out := ULINT_TO_STRING(in);
TryConvert_ULINT_TO_STRING := TRUE;

END_FUNCTION

// mobject-converters/Converters/UDINT_TO_/TryConvert_UDINT_TO_REAL
FUNCTION TryConvert_UDINT_TO_REAL : BOOL
VAR_INPUT
	in : UDINT;
	out : REFERENCE TO REAL;
END_VAR

out := UDINT_TO_REAL(in);
TryConvert_UDINT_TO_REAL := TRUE;

END_FUNCTION

// mobject-converters/Converters/UDINT_TO_/TryConvert_UDINT_TO_LREAL
FUNCTION TryConvert_UDINT_TO_LREAL : BOOL
VAR_INPUT
	in : UDINT;
	out : REFERENCE TO LREAL;
END_VAR

out := UDINT_TO_LREAL(in);
TryConvert_UDINT_TO_LREAL := TRUE;

END_FUNCTION

// mobject-converters/Converters/UDINT_TO_/TryConvert_UDINT_TO_TIME
FUNCTION TryConvert_UDINT_TO_TIME : BOOL
VAR_INPUT
	in : UDINT;
	out : REFERENCE TO TIME;
END_VAR

out := UDINT_TO_TIME(in);
TryConvert_UDINT_TO_TIME := TRUE;

END_FUNCTION

// mobject-converters/Converters/UDINT_TO_/TryConvert_UDINT_TO_TOD
FUNCTION TryConvert_UDINT_TO_TOD : BOOL
VAR_INPUT
	in : UDINT;
	out : REFERENCE TO TOD;
END_VAR

IF in > DatatypeLimits.MAX_VALUE_OF_UDINT_WHICH_CAN_BE_HELD_IN_A_TOD THEN
	RETURN;
END_IF

out := UDINT_TO_TOD(in);
TryConvert_UDINT_TO_TOD := TRUE;

END_FUNCTION

// mobject-converters/Converters/UDINT_TO_/TryConvert_UDINT_TO_DATE
FUNCTION TryConvert_UDINT_TO_DATE : BOOL
VAR_INPUT
	in : UDINT;
	out : REFERENCE TO DATE;
END_VAR

out := UDINT_TO_DATE(in);
TryConvert_UDINT_TO_DATE := TRUE;

END_FUNCTION

// mobject-converters/Converters/UDINT_TO_/TryConvert_UDINT_TO_DT
FUNCTION TryConvert_UDINT_TO_DT : BOOL
VAR_INPUT
	in : UDINT;
	out : REFERENCE TO DT;
END_VAR

out := UDINT_TO_DT(in);
TryConvert_UDINT_TO_DT := TRUE;

END_FUNCTION

// mobject-converters/Converters/UDINT_TO_/TryConvert_UDINT_TO_STRING
FUNCTION TryConvert_UDINT_TO_STRING : BOOL
VAR_INPUT
	in : UDINT;
	out : REFERENCE TO STRING;
END_VAR

out := UDINT_TO_STRING(in);
TryConvert_UDINT_TO_STRING := TRUE;

END_FUNCTION

// mobject-converters/Converters/UINT_TO_/TryConvert_UINT_TO_ULINT
FUNCTION TryConvert_UINT_TO_ULINT : BOOL
VAR_INPUT
	in : UINT;
	out : REFERENCE TO ULINT;
END_VAR

out := UINT_TO_ULINT(in);
TryConvert_UINT_TO_ULINT := TRUE;

END_FUNCTION

// mobject-converters/Converters/UINT_TO_/TryConvert_UINT_TO_REAL
FUNCTION TryConvert_UINT_TO_REAL : BOOL
VAR_INPUT
	in : UINT;
	out : REFERENCE TO REAL;
END_VAR

out := UINT_TO_REAL(in);
TryConvert_UINT_TO_REAL := TRUE;

END_FUNCTION

// mobject-converters/Converters/UINT_TO_/TryConvert_UINT_TO_LREAL
FUNCTION TryConvert_UINT_TO_LREAL : BOOL
VAR_INPUT
	in : UINT;
	out : REFERENCE TO LREAL;
END_VAR

out := UINT_TO_LREAL(in);
TryConvert_UINT_TO_LREAL := TRUE;

END_FUNCTION

// mobject-converters/Converters/UINT_TO_/TryConvert_UINT_TO_TIME
FUNCTION TryConvert_UINT_TO_TIME : BOOL
VAR_INPUT
	in : UINT;
	out : REFERENCE TO TIME;
END_VAR

out := UINT_TO_TIME(in);
TryConvert_UINT_TO_TIME := TRUE;

END_FUNCTION

// mobject-converters/Converters/UINT_TO_/TryConvert_UINT_TO_TOD
FUNCTION TryConvert_UINT_TO_TOD : BOOL
VAR_INPUT
	in : UINT;
	out : REFERENCE TO TOD;
END_VAR

out := UINT_TO_TOD(in);
TryConvert_UINT_TO_TOD := TRUE;

END_FUNCTION

// mobject-converters/Converters/UINT_TO_/TryConvert_UINT_TO_DATE
FUNCTION TryConvert_UINT_TO_DATE : BOOL
VAR_INPUT
	in : UINT;
	out : REFERENCE TO DATE;
END_VAR

out := UINT_TO_DATE(in);
TryConvert_UINT_TO_DATE := TRUE;

END_FUNCTION

// mobject-converters/Converters/UINT_TO_/TryConvert_UINT_TO_DT
FUNCTION TryConvert_UINT_TO_DT : BOOL
VAR_INPUT
	in : UINT;
	out : REFERENCE TO DT;
END_VAR

out := UINT_TO_DT(in);
TryConvert_UINT_TO_DT := TRUE;

END_FUNCTION

// mobject-converters/Converters/UINT_TO_/TryConvert_UINT_TO_STRING
FUNCTION TryConvert_UINT_TO_STRING : BOOL
VAR_INPUT
	in : UINT;
	out : REFERENCE TO STRING;
END_VAR

out := UINT_TO_STRING(in);
TryConvert_UINT_TO_STRING := TRUE;

END_FUNCTION

// mobject-converters/Converters/USINT_TO_/TryConvert_USINT_TO_UDINT
FUNCTION TryConvert_USINT_TO_UDINT : BOOL
VAR_INPUT
	in : USINT;
	out : REFERENCE TO UDINT;
END_VAR

out := USINT_TO_UDINT(in);
TryConvert_USINT_TO_UDINT := TRUE;

END_FUNCTION

// mobject-converters/Converters/USINT_TO_/TryConvert_USINT_TO_ULINT
FUNCTION TryConvert_USINT_TO_ULINT : BOOL
VAR_INPUT
	in : USINT;
	out : REFERENCE TO ULINT;
END_VAR

out := USINT_TO_ULINT(in);
TryConvert_USINT_TO_ULINT := TRUE;

END_FUNCTION

// mobject-converters/Converters/USINT_TO_/TryConvert_USINT_TO_REAL
FUNCTION TryConvert_USINT_TO_REAL : BOOL
VAR_INPUT
	in : USINT;
	out : REFERENCE TO REAL;
END_VAR

out := USINT_TO_REAL(in);
TryConvert_USINT_TO_REAL := TRUE;

END_FUNCTION

// mobject-converters/Converters/USINT_TO_/TryConvert_USINT_TO_LREAL
FUNCTION TryConvert_USINT_TO_LREAL : BOOL
VAR_INPUT
	in : USINT;
	out : REFERENCE TO LREAL;
END_VAR

out := USINT_TO_LREAL(in);
TryConvert_USINT_TO_LREAL := TRUE;

END_FUNCTION

// mobject-converters/Converters/USINT_TO_/TryConvert_USINT_TO_TIME
FUNCTION TryConvert_USINT_TO_TIME : BOOL
VAR_INPUT
	in : USINT;
	out : REFERENCE TO TIME;
END_VAR

out := USINT_TO_TIME(in);
TryConvert_USINT_TO_TIME := TRUE;

END_FUNCTION

// mobject-converters/Converters/USINT_TO_/TryConvert_USINT_TO_TOD
FUNCTION TryConvert_USINT_TO_TOD : BOOL
VAR_INPUT
	in : USINT;
	out : REFERENCE TO TOD;
END_VAR

out := USINT_TO_TOD(in);
TryConvert_USINT_TO_TOD := TRUE;

END_FUNCTION

// mobject-converters/Converters/USINT_TO_/TryConvert_USINT_TO_DATE
FUNCTION TryConvert_USINT_TO_DATE : BOOL
VAR_INPUT
	in : USINT;
	out : REFERENCE TO DATE;
END_VAR

out := USINT_TO_DATE(in);
TryConvert_USINT_TO_DATE := TRUE;

END_FUNCTION

// mobject-converters/Converters/USINT_TO_/TryConvert_USINT_TO_DT
FUNCTION TryConvert_USINT_TO_DT : BOOL
VAR_INPUT
	in : USINT;
	out : REFERENCE TO DT;
END_VAR

out := USINT_TO_DT(in);
TryConvert_USINT_TO_DT := TRUE;

END_FUNCTION

// mobject-converters/Converters/USINT_TO_/TryConvert_USINT_TO_STRING
FUNCTION TryConvert_USINT_TO_STRING : BOOL
VAR_INPUT
	in : USINT;
	out : REFERENCE TO STRING;
END_VAR

out := USINT_TO_STRING(in);
TryConvert_USINT_TO_STRING := TRUE;

END_FUNCTION

// mobject-converters/Converters/LINT_TO_/TryConvert_LINT_TO_UINT
FUNCTION TryConvert_LINT_TO_UINT : BOOL
VAR_INPUT
	in : LINT;
	out : REFERENCE TO UINT;
END_VAR

IF in > DatatypeLimits.MAX_VALUE_OF_LINT_WHICH_CAN_BE_HELD_IN_A_UINT THEN
	RETURN;
END_IF

IF in < DatatypeLimits.MIN_VALUE_OF_LINT_WHICH_CAN_BE_HELD_IN_A_UINT THEN
	RETURN;
END_IF

out := LINT_TO_UINT(in);
TryConvert_LINT_TO_UINT := TRUE;

END_FUNCTION

// mobject-converters/Converters/LINT_TO_/TryConvert_LINT_TO_UDINT
FUNCTION TryConvert_LINT_TO_UDINT : BOOL
VAR_INPUT
	in : LINT;
	out : REFERENCE TO UDINT;
END_VAR

IF in > DatatypeLimits.MAX_VALUE_OF_LINT_WHICH_CAN_BE_HELD_IN_A_UDINT THEN
	RETURN;
END_IF

IF in < DatatypeLimits.MIN_VALUE_OF_LINT_WHICH_CAN_BE_HELD_IN_A_UDINT THEN
	RETURN;
END_IF

out := LINT_TO_UDINT(in);
TryConvert_LINT_TO_UDINT := TRUE;

END_FUNCTION

// mobject-converters/Converters/LINT_TO_/TryConvert_LINT_TO_ULINT
FUNCTION TryConvert_LINT_TO_ULINT : BOOL
VAR_INPUT
	in : LINT;
	out : REFERENCE TO ULINT;
END_VAR

IF in < DatatypeLimits.MIN_VALUE_OF_LINT_WHICH_CAN_BE_HELD_IN_A_ULINT THEN
	RETURN;
END_IF

out := LINT_TO_ULINT(in);
TryConvert_LINT_TO_ULINT := TRUE;

END_FUNCTION

// mobject-converters/Converters/LINT_TO_/TryConvert_LINT_TO_REAL
FUNCTION TryConvert_LINT_TO_REAL : BOOL
VAR_INPUT
	in : LINT;
	out : REFERENCE TO REAL;
END_VAR

out := LINT_TO_REAL(in);
TryConvert_LINT_TO_REAL := TRUE;

END_FUNCTION

// mobject-converters/Converters/LINT_TO_/TryConvert_LINT_TO_LREAL
FUNCTION TryConvert_LINT_TO_LREAL : BOOL
VAR_INPUT
	in : LINT;
	out : REFERENCE TO LREAL;
END_VAR

out := LINT_TO_LREAL(in);
TryConvert_LINT_TO_LREAL := TRUE;

END_FUNCTION

// mobject-converters/Converters/LINT_TO_/TryConvert_LINT_TO_TIME
FUNCTION TryConvert_LINT_TO_TIME : BOOL
VAR_INPUT
	in : LINT;
	out : REFERENCE TO TIME;
END_VAR

IF in > DatatypeLimits.MAX_VALUE_OF_LINT_WHICH_CAN_BE_HELD_IN_A_TIME THEN
	RETURN;
END_IF

IF in < DatatypeLimits.MIN_VALUE_OF_LINT_WHICH_CAN_BE_HELD_IN_A_TIME THEN
	RETURN;
END_IF

out := LINT_TO_TIME(in);
TryConvert_LINT_TO_TIME := TRUE;

END_FUNCTION

// mobject-converters/Converters/LINT_TO_/TryConvert_LINT_TO_TOD
FUNCTION TryConvert_LINT_TO_TOD : BOOL
VAR_INPUT
	in : LINT;
	out : REFERENCE TO TOD;
END_VAR

IF in > DatatypeLimits.MAX_VALUE_OF_LINT_WHICH_CAN_BE_HELD_IN_A_TOD THEN
	RETURN;
END_IF

IF in < DatatypeLimits.MIN_VALUE_OF_LINT_WHICH_CAN_BE_HELD_IN_A_TOD THEN
	RETURN;
END_IF

out := LINT_TO_TOD(in);
TryConvert_LINT_TO_TOD := TRUE;

END_FUNCTION

// mobject-converters/Converters/LINT_TO_/TryConvert_LINT_TO_DATE
FUNCTION TryConvert_LINT_TO_DATE : BOOL
VAR_INPUT
	in : LINT;
	out : REFERENCE TO DATE;
END_VAR

IF in > DatatypeLimits.MAX_VALUE_OF_LINT_WHICH_CAN_BE_HELD_IN_A_DATE THEN
	RETURN;
END_IF

IF in < DatatypeLimits.MIN_VALUE_OF_LINT_WHICH_CAN_BE_HELD_IN_A_DATE THEN
	RETURN;
END_IF

out := LINT_TO_DATE(in);
TryConvert_LINT_TO_DATE := TRUE;

END_FUNCTION

// mobject-converters/Converters/LINT_TO_/TryConvert_LINT_TO_DT
FUNCTION TryConvert_LINT_TO_DT : BOOL
VAR_INPUT
	in : LINT;
	out : REFERENCE TO DT;
END_VAR

IF in > DatatypeLimits.MAX_VALUE_OF_LINT_WHICH_CAN_BE_HELD_IN_A_DT THEN
	RETURN;
END_IF

IF in < DatatypeLimits.MIN_VALUE_OF_LINT_WHICH_CAN_BE_HELD_IN_A_DT THEN
	RETURN;
END_IF

out := LINT_TO_DT(in);
TryConvert_LINT_TO_DT := TRUE;

END_FUNCTION

// mobject-converters/Converters/LINT_TO_/TryConvert_LINT_TO_STRING
FUNCTION TryConvert_LINT_TO_STRING : BOOL
VAR_INPUT
	in : LINT;
	out : REFERENCE TO STRING;
END_VAR

out := LINT_TO_STRING(in);
TryConvert_LINT_TO_STRING := TRUE;

END_FUNCTION

// mobject-converters/Converters/DINT_TO_/TryConvert_DINT_TO_USINT
FUNCTION TryConvert_DINT_TO_USINT : BOOL
VAR_INPUT
	in : DINT;
	out : REFERENCE TO USINT;
END_VAR

IF in > DatatypeLimits.MAX_VALUE_OF_DINT_WHICH_CAN_BE_HELD_IN_A_USINT THEN
	RETURN;
END_IF

IF in < DatatypeLimits.MIN_VALUE_OF_DINT_WHICH_CAN_BE_HELD_IN_A_USINT THEN
	RETURN;
END_IF

out := DINT_TO_USINT(in);
TryConvert_DINT_TO_USINT := TRUE;

END_FUNCTION

// mobject-converters/Converters/DINT_TO_/TryConvert_DINT_TO_UINT
FUNCTION TryConvert_DINT_TO_UINT : BOOL
VAR_INPUT
	in : DINT;
	out : REFERENCE TO UINT;
END_VAR

IF in > DatatypeLimits.MAX_VALUE_OF_DINT_WHICH_CAN_BE_HELD_IN_A_UINT THEN
	RETURN;
END_IF

IF in < DatatypeLimits.MIN_VALUE_OF_DINT_WHICH_CAN_BE_HELD_IN_A_UINT THEN
	RETURN;
END_IF

out := DINT_TO_UINT(in);
TryConvert_DINT_TO_UINT := TRUE;

END_FUNCTION

// mobject-converters/Converters/DINT_TO_/TryConvert_DINT_TO_UDINT
FUNCTION TryConvert_DINT_TO_UDINT : BOOL
VAR_INPUT
	in : DINT;
	out : REFERENCE TO UDINT;
END_VAR

IF in < DatatypeLimits.MIN_VALUE_OF_DINT_WHICH_CAN_BE_HELD_IN_A_UDINT THEN
	RETURN;
END_IF

out := DINT_TO_UDINT(in);
TryConvert_DINT_TO_UDINT := TRUE;

END_FUNCTION

// mobject-converters/Converters/DINT_TO_/TryConvert_DINT_TO_ULINT
FUNCTION TryConvert_DINT_TO_ULINT : BOOL
VAR_INPUT
	in : DINT;
	out : REFERENCE TO ULINT;
END_VAR

IF in < DatatypeLimits.MIN_VALUE_OF_DINT_WHICH_CAN_BE_HELD_IN_A_ULINT THEN
	RETURN;
END_IF

out := DINT_TO_ULINT(in);
TryConvert_DINT_TO_ULINT := TRUE;

END_FUNCTION

// mobject-converters/Converters/DINT_TO_/TryConvert_DINT_TO_REAL
FUNCTION TryConvert_DINT_TO_REAL : BOOL
VAR_INPUT
	in : DINT;
	out : REFERENCE TO REAL;
END_VAR

out := DINT_TO_REAL(in);
TryConvert_DINT_TO_REAL := TRUE;

END_FUNCTION

// mobject-converters/Converters/DINT_TO_/TryConvert_DINT_TO_LREAL
FUNCTION TryConvert_DINT_TO_LREAL : BOOL
VAR_INPUT
	in : DINT;
	out : REFERENCE TO LREAL;
END_VAR

out := DINT_TO_LREAL(in);
TryConvert_DINT_TO_LREAL := TRUE;

END_FUNCTION

// mobject-converters/Converters/DINT_TO_/TryConvert_DINT_TO_TIME
FUNCTION TryConvert_DINT_TO_TIME : BOOL
VAR_INPUT
	in : DINT;
	out : REFERENCE TO TIME;
END_VAR

IF in < DatatypeLimits.MIN_VALUE_OF_DINT_WHICH_CAN_BE_HELD_IN_A_TIME THEN
	RETURN;
END_IF

out := DINT_TO_TIME(in);
TryConvert_DINT_TO_TIME := TRUE;

END_FUNCTION

// mobject-converters/Converters/DINT_TO_/TryConvert_DINT_TO_TOD
FUNCTION TryConvert_DINT_TO_TOD : BOOL
VAR_INPUT
	in : DINT;
	out : REFERENCE TO TOD;
END_VAR

IF in > DatatypeLimits.MAX_VALUE_OF_DINT_WHICH_CAN_BE_HELD_IN_A_TOD THEN
	RETURN;
END_IF

IF in < DatatypeLimits.MIN_VALUE_OF_DINT_WHICH_CAN_BE_HELD_IN_A_TOD THEN
	RETURN;
END_IF

out := DINT_TO_TOD(in);
TryConvert_DINT_TO_TOD := TRUE;

END_FUNCTION

// mobject-converters/Converters/DINT_TO_/TryConvert_DINT_TO_DATE
FUNCTION TryConvert_DINT_TO_DATE : BOOL
VAR_INPUT
	in : DINT;
	out : REFERENCE TO DATE;
END_VAR

IF in < DatatypeLimits.MIN_VALUE_OF_DINT_WHICH_CAN_BE_HELD_IN_A_DATE THEN
	RETURN;
END_IF

out := DINT_TO_DATE(in);
TryConvert_DINT_TO_DATE := TRUE;

END_FUNCTION

// mobject-converters/Converters/DINT_TO_/TryConvert_DINT_TO_DT
FUNCTION TryConvert_DINT_TO_DT : BOOL
VAR_INPUT
	in : DINT;
	out : REFERENCE TO DT;
END_VAR

IF in < DatatypeLimits.MIN_VALUE_OF_DINT_WHICH_CAN_BE_HELD_IN_A_DT THEN
	RETURN;
END_IF

out := DINT_TO_DT(in);
TryConvert_DINT_TO_DT := TRUE;

END_FUNCTION

// mobject-converters/Converters/DINT_TO_/TryConvert_DINT_TO_STRING
FUNCTION TryConvert_DINT_TO_STRING : BOOL
VAR_INPUT
	in : DINT;
	out : REFERENCE TO STRING;
END_VAR

out := DINT_TO_STRING(in);
TryConvert_DINT_TO_STRING := TRUE;

END_FUNCTION

// mobject-converters/Converters/INT_TO_/TryConvert_INT_TO_LINT
FUNCTION TryConvert_INT_TO_LINT : BOOL
VAR_INPUT
	in : INT;
	out : REFERENCE TO LINT;
END_VAR

out := INT_TO_LINT(in);
TryConvert_INT_TO_LINT := TRUE;

END_FUNCTION

// mobject-converters/Converters/INT_TO_/TryConvert_INT_TO_USINT
FUNCTION TryConvert_INT_TO_USINT : BOOL
VAR_INPUT
	in : INT;
	out : REFERENCE TO USINT;
END_VAR

IF in > DatatypeLimits.MAX_VALUE_OF_INT_WHICH_CAN_BE_HELD_IN_A_USINT THEN
	RETURN;
END_IF

IF in < DatatypeLimits.MIN_VALUE_OF_INT_WHICH_CAN_BE_HELD_IN_A_USINT THEN
	RETURN;
END_IF

out := INT_TO_USINT(in);
TryConvert_INT_TO_USINT := TRUE;

END_FUNCTION

// mobject-converters/Converters/INT_TO_/TryConvert_INT_TO_UINT
FUNCTION TryConvert_INT_TO_UINT : BOOL
VAR_INPUT
	in : INT;
	out : REFERENCE TO UINT;
END_VAR

IF in < DatatypeLimits.MIN_VALUE_OF_INT_WHICH_CAN_BE_HELD_IN_A_UINT THEN
	RETURN;
END_IF

out := INT_TO_UINT(in);
TryConvert_INT_TO_UINT := TRUE;

END_FUNCTION

// mobject-converters/Converters/INT_TO_/TryConvert_INT_TO_UDINT
FUNCTION TryConvert_INT_TO_UDINT : BOOL
VAR_INPUT
	in : INT;
	out : REFERENCE TO UDINT;
END_VAR

IF in < DatatypeLimits.MIN_VALUE_OF_INT_WHICH_CAN_BE_HELD_IN_A_UDINT THEN
	RETURN;
END_IF

out := INT_TO_UDINT(in);
TryConvert_INT_TO_UDINT := TRUE;

END_FUNCTION

// mobject-converters/Converters/INT_TO_/TryConvert_INT_TO_ULINT
FUNCTION TryConvert_INT_TO_ULINT : BOOL
VAR_INPUT
	in : INT;
	out : REFERENCE TO ULINT;
END_VAR

IF in < DatatypeLimits.MIN_VALUE_OF_INT_WHICH_CAN_BE_HELD_IN_A_ULINT THEN
	RETURN;
END_IF

out := INT_TO_ULINT(in);
TryConvert_INT_TO_ULINT := TRUE;

END_FUNCTION

// mobject-converters/Converters/INT_TO_/TryConvert_INT_TO_REAL
FUNCTION TryConvert_INT_TO_REAL : BOOL
VAR_INPUT
	in : INT;
	out : REFERENCE TO REAL;
END_VAR

out := INT_TO_REAL(in);
TryConvert_INT_TO_REAL := TRUE;

END_FUNCTION

// mobject-converters/Converters/INT_TO_/TryConvert_INT_TO_LREAL
FUNCTION TryConvert_INT_TO_LREAL : BOOL
VAR_INPUT
	in : INT;
	out : REFERENCE TO LREAL;
END_VAR

out := INT_TO_LREAL(in);
TryConvert_INT_TO_LREAL := TRUE;

END_FUNCTION

// mobject-converters/Converters/INT_TO_/TryConvert_INT_TO_TIME
FUNCTION TryConvert_INT_TO_TIME : BOOL
VAR_INPUT
	in : INT;
	out : REFERENCE TO TIME;
END_VAR

IF in < DatatypeLimits.MIN_VALUE_OF_INT_WHICH_CAN_BE_HELD_IN_A_TIME THEN
	RETURN;
END_IF

out := INT_TO_TIME(in);
TryConvert_INT_TO_TIME := TRUE;

END_FUNCTION

// mobject-converters/Converters/INT_TO_/TryConvert_INT_TO_TOD
FUNCTION TryConvert_INT_TO_TOD : BOOL
VAR_INPUT
	in : INT;
	out : REFERENCE TO TOD;
END_VAR

IF in < DatatypeLimits.MIN_VALUE_OF_INT_WHICH_CAN_BE_HELD_IN_A_TOD THEN
	RETURN;
END_IF

out := INT_TO_TOD(in);
TryConvert_INT_TO_TOD := TRUE;

END_FUNCTION

// mobject-converters/Converters/INT_TO_/TryConvert_INT_TO_DATE
FUNCTION TryConvert_INT_TO_DATE : BOOL
VAR_INPUT
	in : INT;
	out : REFERENCE TO DATE;
END_VAR

IF in < DatatypeLimits.MIN_VALUE_OF_INT_WHICH_CAN_BE_HELD_IN_A_DATE THEN
	RETURN;
END_IF

out := INT_TO_DATE(in);
TryConvert_INT_TO_DATE := TRUE;

END_FUNCTION

// mobject-converters/Converters/INT_TO_/TryConvert_INT_TO_DT
FUNCTION TryConvert_INT_TO_DT : BOOL
VAR_INPUT
	in : INT;
	out : REFERENCE TO DT;
END_VAR

IF in < DatatypeLimits.MIN_VALUE_OF_INT_WHICH_CAN_BE_HELD_IN_A_DT THEN
	RETURN;
END_IF

out := INT_TO_DT(in);
TryConvert_INT_TO_DT := TRUE;

END_FUNCTION

// mobject-converters/Converters/INT_TO_/TryConvert_INT_TO_STRING
FUNCTION TryConvert_INT_TO_STRING : BOOL
VAR_INPUT
	in : INT;
	out : REFERENCE TO STRING;
END_VAR

out := INT_TO_STRING(in);
TryConvert_INT_TO_STRING := TRUE;

END_FUNCTION

// mobject-converters/Converters/SINT_TO_/TryConvert_SINT_TO_DINT
FUNCTION TryConvert_SINT_TO_DINT : BOOL
VAR_INPUT
	in : SINT;
	out : REFERENCE TO DINT;
END_VAR

out := SINT_TO_DINT(in);
TryConvert_SINT_TO_DINT := TRUE;

END_FUNCTION

// mobject-converters/Converters/SINT_TO_/TryConvert_SINT_TO_LINT
FUNCTION TryConvert_SINT_TO_LINT : BOOL
VAR_INPUT
	in : SINT;
	out : REFERENCE TO LINT;
END_VAR

out := SINT_TO_LINT(in);
TryConvert_SINT_TO_LINT := TRUE;

END_FUNCTION

// mobject-converters/Converters/SINT_TO_/TryConvert_SINT_TO_USINT
FUNCTION TryConvert_SINT_TO_USINT : BOOL
VAR_INPUT
	in : SINT;
	out : REFERENCE TO USINT;
END_VAR

IF in < DatatypeLimits.MIN_VALUE_OF_SINT_WHICH_CAN_BE_HELD_IN_A_USINT THEN
	RETURN;
END_IF

out := SINT_TO_USINT(in);
TryConvert_SINT_TO_USINT := TRUE;

END_FUNCTION

// mobject-converters/Converters/SINT_TO_/TryConvert_SINT_TO_UINT
FUNCTION TryConvert_SINT_TO_UINT : BOOL
VAR_INPUT
	in : SINT;
	out : REFERENCE TO UINT;
END_VAR

IF in < DatatypeLimits.MIN_VALUE_OF_SINT_WHICH_CAN_BE_HELD_IN_A_UINT THEN
	RETURN;
END_IF

out := SINT_TO_UINT(in);
TryConvert_SINT_TO_UINT := TRUE;

END_FUNCTION

// mobject-converters/Converters/SINT_TO_/TryConvert_SINT_TO_UDINT
FUNCTION TryConvert_SINT_TO_UDINT : BOOL
VAR_INPUT
	in : SINT;
	out : REFERENCE TO UDINT;
END_VAR

IF in < DatatypeLimits.MIN_VALUE_OF_SINT_WHICH_CAN_BE_HELD_IN_A_UDINT THEN
	RETURN;
END_IF

out := SINT_TO_UDINT(in);
TryConvert_SINT_TO_UDINT := TRUE;

END_FUNCTION

// mobject-converters/Converters/SINT_TO_/TryConvert_SINT_TO_ULINT
FUNCTION TryConvert_SINT_TO_ULINT : BOOL
VAR_INPUT
	in : SINT;
	out : REFERENCE TO ULINT;
END_VAR

IF in < DatatypeLimits.MIN_VALUE_OF_SINT_WHICH_CAN_BE_HELD_IN_A_ULINT THEN
	RETURN;
END_IF

out := SINT_TO_ULINT(in);
TryConvert_SINT_TO_ULINT := TRUE;

END_FUNCTION

// mobject-converters/Converters/SINT_TO_/TryConvert_SINT_TO_REAL
FUNCTION TryConvert_SINT_TO_REAL : BOOL
VAR_INPUT
	in : SINT;
	out : REFERENCE TO REAL;
END_VAR

out := SINT_TO_REAL(in);
TryConvert_SINT_TO_REAL := TRUE;

END_FUNCTION

// mobject-converters/Converters/SINT_TO_/TryConvert_SINT_TO_LREAL
FUNCTION TryConvert_SINT_TO_LREAL : BOOL
VAR_INPUT
	in : SINT;
	out : REFERENCE TO LREAL;
END_VAR

out := SINT_TO_LREAL(in);
TryConvert_SINT_TO_LREAL := TRUE;

END_FUNCTION

// mobject-converters/Converters/SINT_TO_/TryConvert_SINT_TO_TIME
FUNCTION TryConvert_SINT_TO_TIME : BOOL
VAR_INPUT
	in : SINT;
	out : REFERENCE TO TIME;
END_VAR

IF in < DatatypeLimits.MIN_VALUE_OF_SINT_WHICH_CAN_BE_HELD_IN_A_TIME THEN
	RETURN;
END_IF

out := SINT_TO_TIME(in);
TryConvert_SINT_TO_TIME := TRUE;

END_FUNCTION

// mobject-converters/Converters/SINT_TO_/TryConvert_SINT_TO_TOD
FUNCTION TryConvert_SINT_TO_TOD : BOOL
VAR_INPUT
	in : SINT;
	out : REFERENCE TO TOD;
END_VAR

IF in < DatatypeLimits.MIN_VALUE_OF_SINT_WHICH_CAN_BE_HELD_IN_A_TOD THEN
	RETURN;
END_IF

out := SINT_TO_TOD(in);
TryConvert_SINT_TO_TOD := TRUE;

END_FUNCTION

// mobject-converters/Converters/SINT_TO_/TryConvert_SINT_TO_DATE
FUNCTION TryConvert_SINT_TO_DATE : BOOL
VAR_INPUT
	in : SINT;
	out : REFERENCE TO DATE;
END_VAR

IF in < DatatypeLimits.MIN_VALUE_OF_SINT_WHICH_CAN_BE_HELD_IN_A_DATE THEN
	RETURN;
END_IF

out := SINT_TO_DATE(in);
TryConvert_SINT_TO_DATE := TRUE;

END_FUNCTION

// mobject-converters/Converters/SINT_TO_/TryConvert_SINT_TO_DT
FUNCTION TryConvert_SINT_TO_DT : BOOL
VAR_INPUT
	in : SINT;
	out : REFERENCE TO DT;
END_VAR

IF in < DatatypeLimits.MIN_VALUE_OF_SINT_WHICH_CAN_BE_HELD_IN_A_DT THEN
	RETURN;
END_IF

out := SINT_TO_DT(in);
TryConvert_SINT_TO_DT := TRUE;

END_FUNCTION

// mobject-converters/Converters/SINT_TO_/TryConvert_SINT_TO_STRING
FUNCTION TryConvert_SINT_TO_STRING : BOOL
VAR_INPUT
	in : SINT;
	out : REFERENCE TO STRING;
END_VAR

out := SINT_TO_STRING(in);
TryConvert_SINT_TO_STRING := TRUE;

END_FUNCTION

// mobject-converters/Converters/LWORD_TO_/TryConvert_LWORD_TO_INT
FUNCTION TryConvert_LWORD_TO_INT : BOOL
VAR_INPUT
	in : LWORD;
	out : REFERENCE TO INT;
END_VAR

IF in > DatatypeLimits.MAX_VALUE_OF_LWORD_WHICH_CAN_BE_HELD_IN_A_INT THEN
	RETURN;
END_IF

out := LWORD_TO_INT(in);
TryConvert_LWORD_TO_INT := TRUE;

END_FUNCTION

// mobject-converters/Converters/LWORD_TO_/TryConvert_LWORD_TO_DINT
FUNCTION TryConvert_LWORD_TO_DINT : BOOL
VAR_INPUT
	in : LWORD;
	out : REFERENCE TO DINT;
END_VAR

IF in > DatatypeLimits.MAX_VALUE_OF_LWORD_WHICH_CAN_BE_HELD_IN_A_DINT THEN
	RETURN;
END_IF

out := LWORD_TO_DINT(in);
TryConvert_LWORD_TO_DINT := TRUE;

END_FUNCTION

// mobject-converters/Converters/LWORD_TO_/TryConvert_LWORD_TO_LINT
FUNCTION TryConvert_LWORD_TO_LINT : BOOL
VAR_INPUT
	in : LWORD;
	out : REFERENCE TO LINT;
END_VAR

IF in > DatatypeLimits.MAX_VALUE_OF_LWORD_WHICH_CAN_BE_HELD_IN_A_LINT THEN
	RETURN;
END_IF

out := LWORD_TO_LINT(in);
TryConvert_LWORD_TO_LINT := TRUE;

END_FUNCTION

// mobject-converters/Converters/LWORD_TO_/TryConvert_LWORD_TO_USINT
FUNCTION TryConvert_LWORD_TO_USINT : BOOL
VAR_INPUT
	in : LWORD;
	out : REFERENCE TO USINT;
END_VAR

IF in > DatatypeLimits.MAX_VALUE_OF_LWORD_WHICH_CAN_BE_HELD_IN_A_USINT THEN
	RETURN;
END_IF

out := LWORD_TO_USINT(in);
TryConvert_LWORD_TO_USINT := TRUE;

END_FUNCTION

// mobject-converters/Converters/LWORD_TO_/TryConvert_LWORD_TO_UINT
FUNCTION TryConvert_LWORD_TO_UINT : BOOL
VAR_INPUT
	in : LWORD;
	out : REFERENCE TO UINT;
END_VAR

IF in > DatatypeLimits.MAX_VALUE_OF_LWORD_WHICH_CAN_BE_HELD_IN_A_UINT THEN
	RETURN;
END_IF

out := LWORD_TO_UINT(in);
TryConvert_LWORD_TO_UINT := TRUE;

END_FUNCTION

// mobject-converters/Converters/LWORD_TO_/TryConvert_LWORD_TO_UDINT
FUNCTION TryConvert_LWORD_TO_UDINT : BOOL
VAR_INPUT
	in : LWORD;
	out : REFERENCE TO UDINT;
END_VAR

IF in > DatatypeLimits.MAX_VALUE_OF_LWORD_WHICH_CAN_BE_HELD_IN_A_UDINT THEN
	RETURN;
END_IF

out := LWORD_TO_UDINT(in);
TryConvert_LWORD_TO_UDINT := TRUE;

END_FUNCTION

// mobject-converters/Converters/LWORD_TO_/TryConvert_LWORD_TO_ULINT
FUNCTION TryConvert_LWORD_TO_ULINT : BOOL
VAR_INPUT
	in : LWORD;
	out : REFERENCE TO ULINT;
END_VAR

out := LWORD_TO_ULINT(in);
TryConvert_LWORD_TO_ULINT := TRUE;

END_FUNCTION

// mobject-converters/Converters/LWORD_TO_/TryConvert_LWORD_TO_REAL
FUNCTION TryConvert_LWORD_TO_REAL : BOOL
VAR_INPUT
	in : LWORD;
	out : REFERENCE TO REAL;
END_VAR

out := LWORD_TO_REAL(in);
TryConvert_LWORD_TO_REAL := TRUE;

END_FUNCTION

// mobject-converters/Converters/LWORD_TO_/TryConvert_LWORD_TO_LREAL
FUNCTION TryConvert_LWORD_TO_LREAL : BOOL
VAR_INPUT
	in : LWORD;
	out : REFERENCE TO LREAL;
END_VAR

out := LWORD_TO_LREAL(in);
TryConvert_LWORD_TO_LREAL := TRUE;

END_FUNCTION

// mobject-converters/Converters/LWORD_TO_/TryConvert_LWORD_TO_TIME
FUNCTION TryConvert_LWORD_TO_TIME : BOOL
VAR_INPUT
	in : LWORD;
	out : REFERENCE TO TIME;
END_VAR

IF in > DatatypeLimits.MAX_VALUE_OF_LWORD_WHICH_CAN_BE_HELD_IN_A_TIME THEN
	RETURN;
END_IF

out := LWORD_TO_TIME(in);
TryConvert_LWORD_TO_TIME := TRUE;

END_FUNCTION

// mobject-converters/Converters/LWORD_TO_/TryConvert_LWORD_TO_TOD
FUNCTION TryConvert_LWORD_TO_TOD : BOOL
VAR_INPUT
	in : LWORD;
	out : REFERENCE TO TOD;
END_VAR

IF in > DatatypeLimits.MAX_VALUE_OF_LWORD_WHICH_CAN_BE_HELD_IN_A_TOD THEN
	RETURN;
END_IF

out := LWORD_TO_TOD(in);
TryConvert_LWORD_TO_TOD := TRUE;

END_FUNCTION

// mobject-converters/Converters/LWORD_TO_/TryConvert_LWORD_TO_DATE
FUNCTION TryConvert_LWORD_TO_DATE : BOOL
VAR_INPUT
	in : LWORD;
	out : REFERENCE TO DATE;
END_VAR

IF in > DatatypeLimits.MAX_VALUE_OF_LWORD_WHICH_CAN_BE_HELD_IN_A_DATE THEN
	RETURN;
END_IF

out := LWORD_TO_DATE(in);
TryConvert_LWORD_TO_DATE := TRUE;

END_FUNCTION

// mobject-converters/Converters/LWORD_TO_/TryConvert_LWORD_TO_DT
FUNCTION TryConvert_LWORD_TO_DT : BOOL
VAR_INPUT
	in : LWORD;
	out : REFERENCE TO DT;
END_VAR

IF in > DatatypeLimits.MAX_VALUE_OF_LWORD_WHICH_CAN_BE_HELD_IN_A_DT THEN
	RETURN;
END_IF

out := LWORD_TO_DT(in);
TryConvert_LWORD_TO_DT := TRUE;

END_FUNCTION

// mobject-converters/Converters/LWORD_TO_/TryConvert_LWORD_TO_STRING
FUNCTION TryConvert_LWORD_TO_STRING : BOOL
VAR_INPUT
	in : LWORD;
	out : REFERENCE TO STRING;
END_VAR

out := LWORD_TO_STRING(in);
TryConvert_LWORD_TO_STRING := TRUE;

END_FUNCTION

// mobject-converters/Converters/DWORD_TO_/TryConvert_DWORD_TO_SINT
FUNCTION TryConvert_DWORD_TO_SINT : BOOL
VAR_INPUT
	in : DWORD;
	out : REFERENCE TO SINT;
END_VAR

IF in > DatatypeLimits.MAX_VALUE_OF_DWORD_WHICH_CAN_BE_HELD_IN_A_SINT THEN
	RETURN;
END_IF

out := DWORD_TO_SINT(in);
TryConvert_DWORD_TO_SINT := TRUE;

END_FUNCTION

// mobject-converters/Converters/DWORD_TO_/TryConvert_DWORD_TO_INT
FUNCTION TryConvert_DWORD_TO_INT : BOOL
VAR_INPUT
	in : DWORD;
	out : REFERENCE TO INT;
END_VAR

IF in > DatatypeLimits.MAX_VALUE_OF_DWORD_WHICH_CAN_BE_HELD_IN_A_INT THEN
	RETURN;
END_IF

out := DWORD_TO_INT(in);
TryConvert_DWORD_TO_INT := TRUE;

END_FUNCTION

// mobject-converters/Converters/DWORD_TO_/TryConvert_DWORD_TO_DINT
FUNCTION TryConvert_DWORD_TO_DINT : BOOL
VAR_INPUT
	in : DWORD;
	out : REFERENCE TO DINT;
END_VAR

IF in > DatatypeLimits.MAX_VALUE_OF_DWORD_WHICH_CAN_BE_HELD_IN_A_DINT THEN
	RETURN;
END_IF

out := DWORD_TO_DINT(in);
TryConvert_DWORD_TO_DINT := TRUE;

END_FUNCTION

// mobject-converters/Converters/DWORD_TO_/TryConvert_DWORD_TO_LINT
FUNCTION TryConvert_DWORD_TO_LINT : BOOL
VAR_INPUT
	in : DWORD;
	out : REFERENCE TO LINT;
END_VAR

out := DWORD_TO_LINT(in);
TryConvert_DWORD_TO_LINT := TRUE;

END_FUNCTION

// mobject-converters/Converters/DWORD_TO_/TryConvert_DWORD_TO_USINT
FUNCTION TryConvert_DWORD_TO_USINT : BOOL
VAR_INPUT
	in : DWORD;
	out : REFERENCE TO USINT;
END_VAR

IF in > DatatypeLimits.MAX_VALUE_OF_DWORD_WHICH_CAN_BE_HELD_IN_A_USINT THEN
	RETURN;
END_IF

out := DWORD_TO_USINT(in);
TryConvert_DWORD_TO_USINT := TRUE;

END_FUNCTION

// mobject-converters/Converters/DWORD_TO_/TryConvert_DWORD_TO_UINT
FUNCTION TryConvert_DWORD_TO_UINT : BOOL
VAR_INPUT
	in : DWORD;
	out : REFERENCE TO UINT;
END_VAR

IF in > DatatypeLimits.MAX_VALUE_OF_DWORD_WHICH_CAN_BE_HELD_IN_A_UINT THEN
	RETURN;
END_IF

out := DWORD_TO_UINT(in);
TryConvert_DWORD_TO_UINT := TRUE;

END_FUNCTION

// mobject-converters/Converters/DWORD_TO_/TryConvert_DWORD_TO_UDINT
FUNCTION TryConvert_DWORD_TO_UDINT : BOOL
VAR_INPUT
	in : DWORD;
	out : REFERENCE TO UDINT;
END_VAR

out := DWORD_TO_UDINT(in);
TryConvert_DWORD_TO_UDINT := TRUE;

END_FUNCTION

// mobject-converters/Converters/DWORD_TO_/TryConvert_DWORD_TO_ULINT
FUNCTION TryConvert_DWORD_TO_ULINT : BOOL
VAR_INPUT
	in : DWORD;
	out : REFERENCE TO ULINT;
END_VAR

out := DWORD_TO_ULINT(in);
TryConvert_DWORD_TO_ULINT := TRUE;

END_FUNCTION

// mobject-converters/Converters/DWORD_TO_/TryConvert_DWORD_TO_REAL
FUNCTION TryConvert_DWORD_TO_REAL : BOOL
VAR_INPUT
	in : DWORD;
	out : REFERENCE TO REAL;
END_VAR

out := DWORD_TO_REAL(in);
TryConvert_DWORD_TO_REAL := TRUE;

END_FUNCTION

// mobject-converters/Converters/DWORD_TO_/TryConvert_DWORD_TO_LREAL
FUNCTION TryConvert_DWORD_TO_LREAL : BOOL
VAR_INPUT
	in : DWORD;
	out : REFERENCE TO LREAL;
END_VAR

out := DWORD_TO_LREAL(in);
TryConvert_DWORD_TO_LREAL := TRUE;

END_FUNCTION

// mobject-converters/Converters/DWORD_TO_/TryConvert_DWORD_TO_TIME
FUNCTION TryConvert_DWORD_TO_TIME : BOOL
VAR_INPUT
	in : DWORD;
	out : REFERENCE TO TIME;
END_VAR

out := DWORD_TO_TIME(in);
TryConvert_DWORD_TO_TIME := TRUE;

END_FUNCTION

// mobject-converters/Converters/DWORD_TO_/TryConvert_DWORD_TO_TOD
FUNCTION TryConvert_DWORD_TO_TOD : BOOL
VAR_INPUT
	in : DWORD;
	out : REFERENCE TO TOD;
END_VAR

IF in > DatatypeLimits.MAX_VALUE_OF_DWORD_WHICH_CAN_BE_HELD_IN_A_TOD THEN
	RETURN;
END_IF

out := DWORD_TO_TOD(in);
TryConvert_DWORD_TO_TOD := TRUE;

END_FUNCTION

// mobject-converters/Converters/DWORD_TO_/TryConvert_DWORD_TO_DATE
FUNCTION TryConvert_DWORD_TO_DATE : BOOL
VAR_INPUT
	in : DWORD;
	out : REFERENCE TO DATE;
END_VAR

out := DWORD_TO_DATE(in);
TryConvert_DWORD_TO_DATE := TRUE;

END_FUNCTION

// mobject-converters/Converters/DWORD_TO_/TryConvert_DWORD_TO_DT
FUNCTION TryConvert_DWORD_TO_DT : BOOL
VAR_INPUT
	in : DWORD;
	out : REFERENCE TO DT;
END_VAR

out := DWORD_TO_DT(in);
TryConvert_DWORD_TO_DT := TRUE;

END_FUNCTION

// mobject-converters/Converters/DWORD_TO_/TryConvert_DWORD_TO_STRING
FUNCTION TryConvert_DWORD_TO_STRING : BOOL
VAR_INPUT
	in : DWORD;
	out : REFERENCE TO STRING;
END_VAR

out := DWORD_TO_STRING(in);
TryConvert_DWORD_TO_STRING := TRUE;

END_FUNCTION

// mobject-converters/Converters/WORD_TO_/TryConvert_WORD_TO_LWORD
FUNCTION TryConvert_WORD_TO_LWORD : BOOL
VAR_INPUT
	in : WORD;
	out : REFERENCE TO LWORD;
END_VAR

out := WORD_TO_LWORD(in);
TryConvert_WORD_TO_LWORD := TRUE;

END_FUNCTION

